KUKA KRL program: EPS_2_25694_HR03_A_20260120031654.src

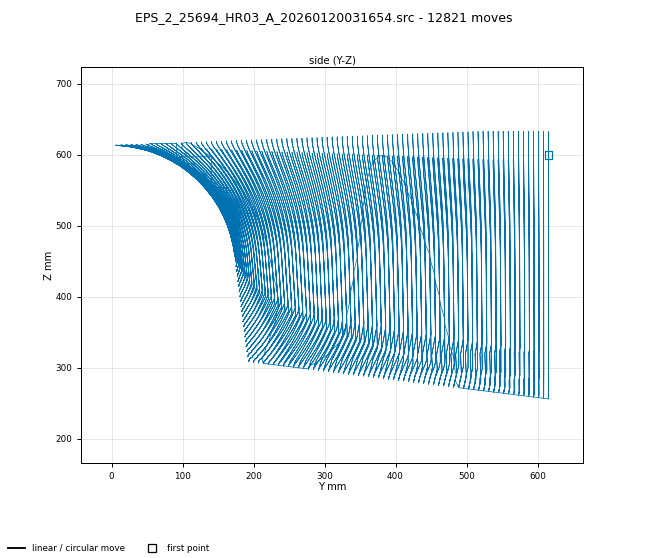
[picture p0: tool path of EPS_2_25694_HR03_A_20260120031654.src, 12821 of 12823 moves have a stored position in this frame; points joined in program order, loops and branches not executed]
&ACCESS RVP
&REL 4
&COMMENT QRS 19112012
&PARAM EDITMASK = *
DEF PART()
EXT BAS (BAS_COMMAND :IN,REAL :IN )
INT I
BAS (#INITMOV,0 )

;KUKA QRS Post kuka4.cps  Date:22-06-2017 !

File_ID=2992

QRS_PRE_INIT()

;Init var - Until changes are made in qrs_pre_init
Outlet_Square_prg=0
Inlet_1_Square_prg=0
Inlet_2_Square_prg=0
Inlet_3_Square_prg=0
Inlet_4_Square_prg=0
Inlet_5_Square_prg=0

Outlet_1={X 0.000, Y 523.550, Z 484.000, B 0.000, E1 0.000 }
Inlet_1={X 0.000, Y 526.470, Z 444.000, B 0.000, E1 180.000 }
Outlet_1_type=299
Inlet_1_type=299
;QRS#1=Sidecore dimensions
;QRS#2=300-12" PVC SDR 35
;QRS#3=300-12" PVC SDR 35
;QRS#4=
;QRS#5=
;QRS#6=
;QRS#7=
;QRS#8=
;QRS#9=16M PSX
;QRS#10=16M PSX
;QRS#11=
;QRS#12=
;QRS#13=
;QRS#14=
;QRS#15=
;QRS#16=1220x127x914 3'
;QRS#17=EPS Height
;QRS#18=633,5
;QRS#19=*
;QRS#20= UPDATED VERSION 22-06-2017
;QRS#21=*
Outlet_Square=0150
Inlet_1_Square=0150
Inlet_2_Square=0
Inlet_3_Square=0
Inlet_4_Square=0
Inlet_5_Square=0
Mill_Square=1
Outlet_Square_Prg=206
Inlet_1_Square_prg=206

QRS_INIT()

$ADVANCE=5

; T1
PTP {E1 173.656,E2 173.656}
PTP {X 0,Y 615.44,A -85,B 0,C 180,E1 173.656,E2 173.656,E3 0,E4 0,E5 0,E6 0}
QRS_SPEED_INIT()
LIN {X 0,Y 615.44,Z 600,A -85,B 0,C 180,E1 173.656,E2 173.656,E3 0,E4 0,E5 0,E6 0} C_VEL
LIN {X 0,Y 615.44,Z 266.5,A -85,B 0,C 180,E1 173.656,E2 173.656} C_VEL
LIN {X 0,Y 615.44,Z 258.32,A -85,B 0,C 180,E1 173.656,E2 173.656} C_VEL
LIN {X 0,Y 615.434,Z 256.32,A -85,B 0,C 180,E1 173.47,E2 173.47} C_VEL
LIN {X 0,Y 615.463,Z 256.318,A -85,B 0,C 180,E1 170.801,E2 170.801} C_VEL
LIN {X 0,Y 615.474,Z 256.325,A -85,B 0,C 180,E1 168.139,E2 168.139} C_VEL
LIN {X 0,Y 615.429,Z 256.321,A -85,B 0,C 180,E1 165.449,E2 165.449} C_VEL
LIN {X 0,Y 615.48,Z 256.318,A -85,B 0,C 180,E1 162.729,E2 162.729} C_VEL
LIN {X 0,Y 615.445,Z 256.323,A -85,B 0,C 180,E1 159.966,E2 159.966} C_VEL
LIN {X 0,Y 615.426,Z 256.322,A -85,B 0,C 180,E1 157.669,E2 157.669} C_VEL
LIN {X 0,Y 615.425,Z 256.323,A -85,B 0,C 180,E1 155.725,E2 155.725} C_VEL
LIN {X 0,Y 615.423,Z 256.322,A -85,B 0,C 180,E1 153.553,E2 153.553} C_VEL
LIN {X 0,Y 615.493,Z 256.324,A -85,B 0,C 180,E1 150.594,E2 150.594} C_VEL
LIN {X 0,Y 615.465,Z 256.324,A -85,B 0,C 180,E1 148.313,E2 148.313} C_VEL
LIN {X 0,Y 615.429,Z 256.324,A -85,B 0,C 180,E1 145.974,E2 145.974} C_VEL
LIN {X 0,Y 615.418,Z 256.323,A -85,B 0,C 180,E1 143.57,E2 143.57} C_VEL
LIN {X 0,Y 615.463,Z 256.323,A -85,B 0,C 180,E1 140.942,E2 140.942} C_VEL
LIN {X 0,Y 615.473,Z 256.326,A -85,B 0,C 180,E1 138.525,E2 138.525} C_VEL
LIN {X 0,Y 615.42,Z 256.325,A -85,B 0,C 180,E1 136.01,E2 136.01} C_VEL
LIN {X 0,Y 615.417,Z 256.325,A -85,B 0,C 180,E1 133.99,E2 133.99} C_VEL
LIN {X 0,Y 615.417,Z 256.325,A -85,B 0,C 180,E1 131.48,E2 131.48} C_VEL
LIN {X 0,Y 615.473,Z 256.327,A -85,B 0,C 180,E1 128.906,E2 128.906} C_VEL
LIN {X 0,Y 615.446,Z 256.324,A -85,B 0,C 180,E1 126.428,E2 126.428} C_VEL
LIN {X 0,Y 615.416,Z 256.324,A -85,B 0,C 180,E1 124.027,E2 124.027} C_VEL
LIN {X 0,Y 615.415,Z 256.325,A -85,B 0,C 180,E1 121.69,E2 121.69} C_VEL
LIN {X 0,Y 615.435,Z 256.324,A -85,B 0,C 180,E1 119.41,E2 119.41} C_VEL
LIN {X 0,Y 615.445,Z 256.322,A -85,B 0,C 180,E1 116.447,E2 116.447} C_VEL
LIN {X 0,Y 615.419,Z 256.323,A -85,B 0,C 180,E1 113.994,E2 113.994} C_VEL
LIN {X 0,Y 615.424,Z 256.408,A -85,B 0,C 180,E1 111.72,E2 111.72} C_VEL
LIN {X 0,Y 615.484,Z 275.615,A -85,B 0,C 180,E1 109.165,E2 109.165} C_VEL
LIN {X 0,Y 615.468,Z 283.1,A -85,B 0,C 180,E1 108.181,E2 108.181} C_VEL
LIN {X 0,Y 615.489,Z 447.324,A -85,B 0,C 180,E1 106.2,E2 106.2} C_VEL
LIN {X 0,Y 615.489,Z 461.801,A -85,B 0,C 180,E1 105.906,E2 105.906} C_VEL
LIN {X 0,Y 615.477,Z 476.406,A -85,B 0,C 180,E1 105.481,E2 105.481} C_VEL
LIN {X 0,Y 615.491,Z 489.73,A -85,B 0,C 180,E1 104.972,E2 104.972} C_VEL
LIN {X 0,Y 615.483,Z 503.376,A -85,B 0,C 180,E1 104.32,E2 104.32} C_VEL
LIN {X 0,Y 615.5,Z 516.661,A -85,B 0,C 180,E1 103.538,E2 103.538} C_VEL
LIN {X 0,Y 615.497,Z 528.512,A -85,B 0,C 180,E1 102.698,E2 102.698} C_VEL
LIN {X 0,Y 615.497,Z 540.356,A -85,B 0,C 180,E1 101.694,E2 101.694} C_VEL
LIN {X 0,Y 615.495,Z 550.165,A -85,B 0,C 180,E1 100.709,E2 100.709} C_VEL
LIN {X 0,Y 615.495,Z 560.01,A -85,B 0,C 180,E1 99.531,E2 99.531} C_VEL
LIN {X 0,Y 615.497,Z 568.101,A -85,B 0,C 180,E1 98.371,E2 98.371} C_VEL
LIN {X 0,Y 615.491,Z 574.781,A -85,B 0,C 180,E1 97.216,E2 97.216} C_VEL
LIN {X 0,Y 615.497,Z 580.947,A -85,B 0,C 180,E1 95.899,E2 95.899} C_VEL
LIN {X 0,Y 615.49,Z 585.715,A -85,B 0,C 180,E1 94.585,E2 94.585} C_VEL
LIN {X 0,Y 615.491,Z 589.22,A -85,B 0,C 180,E1 93.273,E2 93.273} C_VEL
LIN {X 0,Y 615.499,Z 591.539,A -85,B 0,C 180,E1 91.963,E2 91.963} C_VEL
LIN {X 0,Y 615.491,Z 592.728,A -85,B 0,C 180,E1 90.655,E2 90.655} C_VEL
LIN {X 0,Y 615.492,Z 592.751,A -85,B 0,C 180,E1 89.346,E2 89.346} C_VEL
LIN {X 0,Y 615.499,Z 591.646,A -85,B 0,C 180,E1 88.037,E2 88.037} C_VEL
LIN {X 0,Y 615.494,Z 589.416,A -85,B 0,C 180,E1 86.727,E2 86.727} C_VEL
LIN {X 0,Y 615.491,Z 586.006,A -85,B 0,C 180,E1 85.416,E2 85.416} C_VEL
LIN {X 0,Y 615.498,Z 581.337,A -85,B 0,C 180,E1 84.102,E2 84.102} C_VEL
LIN {X 0,Y 615.49,Z 575.273,A -85,B 0,C 180,E1 82.785,E2 82.785} C_VEL
LIN {X 0,Y 615.49,Z 567.635,A -85,B 0,C 180,E1 81.464,E2 81.464} C_VEL
LIN {X 0,Y 615.495,Z 559.452,A -85,B 0,C 180,E1 80.304,E2 80.304} C_VEL
LIN {X 0,Y 615.496,Z 549.333,A -85,B 0,C 180,E1 79.109,E2 79.109} C_VEL
LIN {X 0,Y 615.498,Z 537.685,A -85,B 0,C 180,E1 77.973,E2 77.973} C_VEL
LIN {X 0,Y 615.498,Z 526.415,A -85,B 0,C 180,E1 77.051,E2 77.051} C_VEL
LIN {X 0,Y 615.498,Z 514.177,A -85,B 0,C 180,E1 76.211,E2 76.211} C_VEL
LIN {X 0,Y 615.48,Z 500.78,A -85,B 0,C 180,E1 75.451,E2 75.451} C_VEL
LIN {X 0,Y 615.488,Z 485.866,A -85,B 0,C 180,E1 74.774,E2 74.774} C_VEL
LIN {X 0,Y 615.477,Z 471.391,A -85,B 0,C 180,E1 74.265,E2 74.265} C_VEL
LIN {X 0,Y 615.491,Z 455.809,A -85,B 0,C 180,E1 73.866,E2 73.866} C_VEL
LIN {X 0,Y 615.486,Z 439.601,A -85,B 0,C 180,E1 73.603,E2 73.603} C_VEL
LIN {X 0,Y 615.472,Z 283.019,A -85,B 0,C 180,E1 71.718,E2 71.718} C_VEL
LIN {X 0,Y 615.498,Z 261.851,A -85,B 0,C 180,E1 68.92,E2 68.92} C_VEL
LIN {X 0,Y 615.43,Z 256.322,A -85,B 0,C 180,E1 68.17,E2 68.17} C_VEL
LIN {X 0,Y 615.434,Z 256.32,A -85,B 0,C 180,E1 65.726,E2 65.726} C_VEL
LIN {X 0,Y 615.494,Z 256.326,A -85,B 0,C 180,E1 62.954,E2 62.954} C_VEL
LIN {X 0,Y 615.423,Z 256.323,A -85,B 0,C 180,E1 60.216,E2 60.216} C_VEL
LIN {X 0,Y 615.425,Z 256.323,A -85,B 0,C 180,E1 58.311,E2 58.311} C_VEL
LIN {X 0,Y 615.422,Z 256.322,A -85,B 0,C 180,E1 55.974,E2 55.974} C_VEL
LIN {X 0,Y 615.449,Z 256.322,A -85,B 0,C 180,E1 53.573,E2 53.573} C_VEL
LIN {X 0,Y 615.47,Z 256.325,A -85,B 0,C 180,E1 50.94,E2 50.94} C_VEL
LIN {X 0,Y 615.425,Z 256.324,A -85,B 0,C 180,E1 48.521,E2 48.521} C_VEL
LIN {X 0,Y 615.417,Z 256.324,A -85,B 0,C 180,E1 46.009,E2 46.009} C_VEL
LIN {X 0,Y 615.498,Z 256.325,A -85,B 0,C 180,E1 43.244,E2 43.244} C_VEL
LIN {X 0,Y 615.42,Z 256.325,A -85,B 0,C 180,E1 40.612,E2 40.612} C_VEL
LIN {X 0,Y 615.418,Z 256.325,A -85,B 0,C 180,E1 38.004,E2 38.004} C_VEL
LIN {X 0,Y 615.456,Z 256.325,A -85,B 0,C 180,E1 35.618,E2 35.618} C_VEL
LIN {X 0,Y 615.483,Z 256.324,A -85,B 0,C 180,E1 33.237,E2 33.237} C_VEL
LIN {X 0,Y 615.444,Z 256.323,A -85,B 0,C 180,E1 30.922,E2 30.922} C_VEL
LIN {X 0,Y 615.416,Z 256.323,A -85,B 0,C 180,E1 28.438,E2 28.438} C_VEL
LIN {X 0,Y 615.418,Z 256.323,A -85,B 0,C 180,E1 26.447,E2 26.447} C_VEL
LIN {X 0,Y 615.435,Z 256.324,A -85,B 0,C 180,E1 23.998,E2 23.998} C_VEL
LIN {X 0,Y 615.498,Z 256.322,A -85,B 0,C 180,E1 21.432,E2 21.432} C_VEL
LIN {X 0,Y 615.424,Z 256.322,A -85,B 0,C 180,E1 18.587,E2 18.587} C_VEL
LIN {X 0,Y 615.424,Z 256.322,A -85,B 0,C 180,E1 16.412,E2 16.412} C_VEL
LIN {X 0,Y 615.461,Z 256.325,A -85,B 0,C 180,E1 13.875,E2 13.875} C_VEL
LIN {X 0,Y 615.466,Z 256.318,A -85,B 0,C 180,E1 11.194,E2 11.194} C_VEL
LIN {X 0,Y 615.429,Z 256.321,A -85,B 0,C 180,E1 8.538,E2 8.538} C_VEL
LIN {X 0,Y 615.475,Z 256.324,A -85,B 0,C 180,E1 5.899,E2 5.899} C_VEL
LIN {X 0,Y 615.471,Z 256.317,A -85,B 0,C 180,E1 3.273,E2 3.273} C_VEL
LIN {X 0,Y 615.433,Z 256.32,A -85,B 0,C 180,E1 0.654,E2 0.654} C_VEL
LIN {X 0,Y 615.471,Z 256.324,A -85,B 0,C 180,E1 -1.963,E2 -1.963} C_VEL
LIN {X 0,Y 615.485,Z 256.314,A -85,B 0,C 180,E1 -4.584,E2 -4.584} C_VEL
LIN {X 0,Y 615.438,Z 256.319,A -85,B 0,C 180,E1 -7.216,E2 -7.216} C_VEL
LIN {X 0,Y 615.472,Z 256.324,A -85,B 0,C 180,E1 -9.862,E2 -9.862} C_VEL
LIN {X 0,Y 615.48,Z 256.314,A -85,B 0,C 180,E1 -12.53,E2 -12.53} C_VEL
LIN {X 0,Y 615.441,Z 256.319,A -85,B 0,C 180,E1 -15.227,E2 -15.227} C_VEL
LIN {X 0,Y 615.493,Z 256.326,A -85,B 0,C 180,E1 -17.957,E2 -17.957} C_VEL
LIN {X 0,Y 615.462,Z 256.314,A -85,B 0,C 180,E1 -20.732,E2 -20.732} C_VEL
LIN {X 0,Y 615.454,Z 256.315,A -85,B 0,C 180,E1 -22.846,E2 -22.846} C_VEL
LIN {X 0,Y 615.449,Z 256.316,A -85,B 0,C 180,E1 -24.993,E2 -24.993} C_VEL
LIN {X 0,Y 615.449,Z 256.318,A -85,B 0,C 180,E1 -27.179,E2 -27.179} C_VEL
LIN {X 0,Y 615.498,Z 256.325,A -85,B 0,C 180,E1 -29.797,E2 -29.797} C_VEL
LIN {X 0,Y 615.484,Z 256.31,A -85,B 0,C 180,E1 -32.458,E2 -32.458} C_VEL
LIN {X 0,Y 615.457,Z 256.314,A -85,B 0,C 180,E1 -34.817,E2 -34.817} C_VEL
LIN {X 0,Y 615.458,Z 256.32,A -85,B 0,C 180,E1 -37.244,E2 -37.244} C_VEL
LIN {X 0,Y 615.493,Z 256.313,A -85,B 0,C 180,E1 -40.09,E2 -40.09} C_VEL
LIN {X 0,Y 615.49,Z 256.309,A -85,B 0,C 180,E1 -42.353,E2 -42.353} C_VEL
LIN {X 0,Y 615.459,Z 256.318,A -85,B 0,C 180,E1 -45.071,E2 -45.071} C_VEL
LIN {X 0,Y 615.49,Z 256.316,A -85,B 0,C 180,E1 -47.919,E2 -47.919} C_VEL
LIN {X 0,Y 615.493,Z 256.308,A -85,B 0,C 180,E1 -50.251,E2 -50.251} C_VEL
LIN {X 0,Y 615.465,Z 256.319,A -85,B 0,C 180,E1 -53.066,E2 -53.066} C_VEL
LIN {X 0,Y 615.482,Z 256.322,A -85,B 0,C 180,E1 -55.3,E2 -55.3} C_VEL
LIN {X 0,Y 615.483,Z 256.309,A -85,B 0,C 180,E1 -58.315,E2 -58.315} C_VEL
LIN {X 0,Y 615.468,Z 256.312,A -85,B 0,C 180,E1 -60.593,E2 -60.593} C_VEL
LIN {X 0,Y 615.469,Z 256.318,A -85,B 0,C 180,E1 -62.958,E2 -62.958} C_VEL
LIN {X 0,Y 615.47,Z 256.455,A -85,B 0,C 180,E1 -64.541,E2 -64.541} C_VEL
LIN {X 0,Y 615.483,Z 280.841,A -85,B 0,C 180,E1 -67.28,E2 -67.28} C_VEL
LIN {X 0,Y 615.494,Z 305.255,A -85,B 0,C 180,E1 -69.968,E2 -69.968} C_VEL
LIN {X 0,Y 615.499,Z 322.022,A -85,B 0,C 180,E1 -71.762,E2 -71.762} C_VEL
LIN {X 0,Y 615.487,Z 488.125,A -85,B 0,C 180,E1 -73.767,E2 -73.767} C_VEL
LIN {X 0,Y 615.49,Z 503.724,A -85,B 0,C 180,E1 -74.095,E2 -74.095} C_VEL
LIN {X 0,Y 615.48,Z 519.059,A -85,B 0,C 180,E1 -74.562,E2 -74.562} C_VEL
LIN {X 0,Y 615.492,Z 532.76,A -85,B 0,C 180,E1 -75.113,E2 -75.113} C_VEL
LIN {X 0,Y 615.494,Z 547.048,A -85,B 0,C 180,E1 -75.834,E2 -75.834} C_VEL
LIN {X 0,Y 615.497,Z 559.903,A -85,B 0,C 180,E1 -76.631,E2 -76.631} C_VEL
LIN {X 0,Y 615.495,Z 572.259,A -85,B 0,C 180,E1 -77.554,E2 -77.554} C_VEL
LIN {X 0,Y 615.495,Z 582.61,A -85,B 0,C 180,E1 -78.474,E2 -78.474} C_VEL
LIN {X 0,Y 615.495,Z 592.187,A -85,B 0,C 180,E1 -79.473,E2 -79.473} C_VEL
LIN {X 0,Y 615.494,Z 601.579,A -85,B 0,C 180,E1 -80.636,E2 -80.636} C_VEL
LIN {X 0,Y 615.495,Z 609.383,A -85,B 0,C 180,E1 -81.794,E2 -81.794} C_VEL
LIN {X 0,Y 615.496,Z 616.607,A -85,B 0,C 180,E1 -83.102,E2 -83.102} C_VEL
LIN {X 0,Y 615.499,Z 622.438,A -85,B 0,C 180,E1 -84.431,E2 -84.431} C_VEL
LIN {X 0,Y 615.491,Z 625.861,A -85,B 0,C 180,E1 -85.416,E2 -85.416} C_VEL
LIN {X 0,Y 615.492,Z 629.319,A -85,B 0,C 180,E1 -86.727,E2 -86.727} C_VEL
LIN {X 0,Y 615.497,Z 631.594,A -85,B 0,C 180,E1 -88.037,E2 -88.037} C_VEL
LIN {X 0,Y 615.493,Z 632.741,A -85,B 0,C 180,E1 -89.346,E2 -89.346} C_VEL
LIN {X 0,Y 615.493,Z 632.74,A -85,B 0,C 180,E1 -90.655,E2 -90.655} C_VEL
LIN {X 0,Y 615.497,Z 631.593,A -85,B 0,C 180,E1 -91.963,E2 -91.963} C_VEL
LIN {X 0,Y 615.492,Z 629.317,A -85,B 0,C 180,E1 -93.273,E2 -93.273} C_VEL
LIN {X 0,Y 615.491,Z 625.859,A -85,B 0,C 180,E1 -94.585,E2 -94.585} C_VEL
LIN {X 0,Y 615.49,Z 621.142,A -85,B 0,C 180,E1 -95.899,E2 -95.899} C_VEL
LIN {X 0,Y 615.495,Z 615.027,A -85,B 0,C 180,E1 -97.216,E2 -97.216} C_VEL
LIN {X 0,Y 615.49,Z 607.331,A -85,B 0,C 180,E1 -98.537,E2 -98.537} C_VEL
LIN {X 0,Y 615.495,Z 599.111,A -85,B 0,C 180,E1 -99.696,E2 -99.696} C_VEL
LIN {X 0,Y 615.497,Z 588.895,A -85,B 0,C 180,E1 -100.893,E2 -100.893} C_VEL
LIN {X 0,Y 615.495,Z 579.063,A -85,B 0,C 180,E1 -101.861,E2 -101.861} C_VEL
LIN {X 0,Y 615.498,Z 566.942,A -85,B 0,C 180,E1 -102.866,E2 -102.866} C_VEL
LIN {X 0,Y 615.498,Z 554.792,A -85,B 0,C 180,E1 -103.706,E2 -103.706} C_VEL
LIN {X 0,Y 615.484,Z 541.372,A -85,B 0,C 180,E1 -104.473,E2 -104.473} C_VEL
LIN {X 0,Y 615.495,Z 526.839,A -85,B 0,C 180,E1 -105.141,E2 -105.141} C_VEL
LIN {X 0,Y 615.484,Z 512.604,A -85,B 0,C 180,E1 -105.651,E2 -105.651} C_VEL
LIN {X 0,Y 615.499,Z 498.113,A -85,B 0,C 180,E1 -106.036,E2 -106.036} C_VEL
LIN {X 0,Y 615.487,Z 483.525,A -85,B 0,C 180,E1 -106.298,E2 -106.298} C_VEL
LIN {X 0,Y 615.497,Z 321.596,A -85,B 0,C 180,E1 -108.259,E2 -108.259} C_VEL
LIN {X 0,Y 615.476,Z 295.674,A -85,B 0,C 180,E1 -111.082,E2 -111.082} C_VEL
LIN {X 0,Y 615.495,Z 271.314,A -85,B 0,C 180,E1 -113.782,E2 -113.782} C_VEL
LIN {X 0,Y 615.472,Z 256.311,A -85,B 0,C 180,E1 -115.495,E2 -115.495} C_VEL
LIN {X 0,Y 615.49,Z 256.322,A -85,B 0,C 180,E1 -118.451,E2 -118.451} C_VEL
LIN {X 0,Y 615.464,Z 256.318,A -85,B 0,C 180,E1 -121.082,E2 -121.082} C_VEL
LIN {X 0,Y 615.475,Z 256.31,A -85,B 0,C 180,E1 -123.532,E2 -123.532} C_VEL
LIN {X 0,Y 615.485,Z 256.326,A -85,B 0,C 180,E1 -126.425,E2 -126.425} C_VEL
LIN {X 0,Y 615.461,Z 256.317,A -85,B 0,C 180,E1 -129.059,E2 -129.059} C_VEL
LIN {X 0,Y 615.472,Z 256.311,A -85,B 0,C 180,E1 -131.476,E2 -131.476} C_VEL
LIN {X 0,Y 615.488,Z 256.319,A -85,B 0,C 180,E1 -134.15,E2 -134.15} C_VEL
LIN {X 0,Y 615.466,Z 256.32,A -85,B 0,C 180,E1 -136.754,E2 -136.754} C_VEL
LIN {X 0,Y 615.468,Z 256.312,A -85,B 0,C 180,E1 -139.392,E2 -139.392} C_VEL
LIN {X 0,Y 615.49,Z 256.316,A -85,B 0,C 180,E1 -141.989,E2 -141.989} C_VEL
LIN {X 0,Y 615.488,Z 256.324,A -85,B 0,C 180,E1 -144.384,E2 -144.384} C_VEL
LIN {X 0,Y 615.457,Z 256.319,A -85,B 0,C 180,E1 -146.762,E2 -146.762} C_VEL
LIN {X 0,Y 615.454,Z 256.315,A -85,B 0,C 180,E1 -149.078,E2 -149.078} C_VEL
LIN {X 0,Y 615.487,Z 256.31,A -85,B 0,C 180,E1 -151.551,E2 -151.551} C_VEL
LIN {X 0,Y 615.469,Z 256.322,A -85,B 0,C 180,E1 -154.436,E2 -154.436} C_VEL
LIN {X 0,Y 615.466,Z 256.322,A -85,B 0,C 180,E1 -156.443,E2 -156.443} C_VEL
LIN {X 0,Y 615.456,Z 256.32,A -85,B 0,C 180,E1 -158.567,E2 -158.567} C_VEL
LIN {X 0,Y 615.45,Z 256.319,A -85,B 0,C 180,E1 -160.661,E2 -160.661} C_VEL
LIN {X 0,Y 615.446,Z 256.319,A -85,B 0,C 180,E1 -162.728,E2 -162.728} C_VEL
LIN {X 0,Y 615.483,Z 256.312,A -85,B 0,C 180,E1 -165.451,E2 -165.451} C_VEL
LIN {X 0,Y 615.48,Z 256.324,A -85,B 0,C 180,E1 -168.139,E2 -168.139} C_VEL
LIN {X 0,Y 615.442,Z 256.318,A -85,B 0,C 180,E1 -170.801,E2 -170.801} C_VEL
LIN {X 0,Y 615.487,Z 256.313,A -85,B 0,C 180,E1 -173.443,E2 -173.443} C_VEL
LIN {X 0,Y 615.476,Z 256.324,A -85,B 0,C 180,E1 -176.071,E2 -176.071} C_VEL
LIN {X 0,Y 615.438,Z 256.319,A -85,B 0,C 180,E1 -178.691,E2 -178.691} C_VEL
LIN {X 0,Y 615.475,Z 256.315,A -85,B 0,C 180,E1 -181.309,E2 -181.309} C_VEL
LIN {X 0,Y 615.477,Z 256.325,A -85,B 0,C 180,E1 -183.929,E2 -183.929} C_VEL
LIN {X 0,Y 615.434,Z 256.32,A -85,B 0,C 180,E1 -186.53,E2 -186.53} C_VEL
LIN {X 0,Y 614.778,Z 256.465,A -85,B 0,C 180,E1 -187.076,E2 -187.076} C_VEL
LIN {X 0,Y 611.96,Z 256.882,A -85,B 0,C 180,E1 -187.962,E2 -187.962} C_VEL
LIN {X 0,Y 609.571,Z 257.191,A -85,B 0,C 180,E1 -188.675,E2 -188.675} C_VEL
LIN {X 0,Y 608.534,Z 257.307,A -85,B 0,C 180,E1 -189.225,E2 -189.225} C_VEL
LIN {X 0,Y 608.444,Z 257.317,A -85,B 0,C 180,E1 -189.411,E2 -189.411} C_VEL
LIN {X 0,Y 608.443,Z 257.319,A -85,B 0,C 180,E1 -192,E2 -192} C_VEL
LIN {X 0,Y 608.405,Z 257.318,A -85,B 0,C 180,E1 -194.722,E2 -194.722} C_VEL
LIN {X 0,Y 608.44,Z 257.322,A -85,B 0,C 180,E1 -197.477,E2 -197.477} C_VEL
LIN {X 0,Y 608.416,Z 257.318,A -85,B 0,C 180,E1 -200.276,E2 -200.276} C_VEL
LIN {X 0,Y 608.397,Z 257.319,A -85,B 0,C 180,E1 -202.461,E2 -202.461} C_VEL
LIN {X 0,Y 608.411,Z 257.318,A -85,B 0,C 180,E1 -204.573,E2 -204.573} C_VEL
LIN {X 0,Y 608.463,Z 257.316,A -85,B 0,C 180,E1 -207.203,E2 -207.203} C_VEL
LIN {X 0,Y 608.412,Z 257.32,A -85,B 0,C 180,E1 -209.961,E2 -209.961} C_VEL
LIN {X 0,Y 608.405,Z 257.318,A -85,B 0,C 180,E1 -212.513,E2 -212.513} C_VEL
LIN {X 0,Y 608.406,Z 257.321,A -85,B 0,C 180,E1 -214.899,E2 -214.899} C_VEL
LIN {X 0,Y 608.432,Z 257.319,A -85,B 0,C 180,E1 -217.749,E2 -217.749} C_VEL
LIN {X 0,Y 608.405,Z 257.318,A -85,B 0,C 180,E1 -220.323,E2 -220.323} C_VEL
LIN {X 0,Y 608.426,Z 257.32,A -85,B 0,C 180,E1 -222.962,E2 -222.962} C_VEL
LIN {X 0,Y 608.407,Z 257.321,A -85,B 0,C 180,E1 -225.741,E2 -225.741} C_VEL
LIN {X 0,Y 608.405,Z 257.319,A -85,B 0,C 180,E1 -227.933,E2 -227.933} C_VEL
LIN {X 0,Y 608.413,Z 257.32,A -85,B 0,C 180,E1 -230.709,E2 -230.709} C_VEL
LIN {X 0,Y 608.435,Z 257.324,A -85,B 0,C 180,E1 -233.083,E2 -233.083} C_VEL
LIN {X 0,Y 608.448,Z 257.317,A -85,B 0,C 180,E1 -235.529,E2 -235.529} C_VEL
LIN {X 0,Y 608.414,Z 257.318,A -85,B 0,C 180,E1 -237.902,E2 -237.902} C_VEL
LIN {X 0,Y 608.404,Z 257.319,A -85,B 0,C 180,E1 -240.217,E2 -240.217} C_VEL
LIN {X 0,Y 608.441,Z 257.32,A -85,B 0,C 180,E1 -242.8,E2 -242.8} C_VEL
LIN {X 0,Y 608.428,Z 257.32,A -85,B 0,C 180,E1 -245.427,E2 -245.427} C_VEL
LIN {X 0,Y 608.428,Z 257.399,A -85,B 0,C 180,E1 -248.151,E2 -248.151} C_VEL
LIN {X 0,Y 608.549,Z 271.691,A -85,B 0,C 180,E1 -250.081,E2 -250.081} C_VEL
LIN {X 0,Y 608.517,Z 283.131,A -85,B 0,C 180,E1 -251.604,E2 -251.604} C_VEL
LIN {X 0,Y 608.727,Z 300.004,A -85,B 0,C 180,E1 -251.816,E2 -251.816} C_VEL
LIN {X 0,Y 608.684,Z 448.405,A -85,B 0,C 180,E1 -253.631,E2 -253.631} C_VEL
LIN {X 0,Y 608.648,Z 463.624,A -85,B 0,C 180,E1 -253.954,E2 -253.954} C_VEL
LIN {X 0,Y 608.61,Z 478.983,A -85,B 0,C 180,E1 -254.426,E2 -254.426} C_VEL
LIN {X 0,Y 608.59,Z 493.666,A -85,B 0,C 180,E1 -255.025,E2 -255.025} C_VEL
LIN {X 0,Y 608.571,Z 507.434,A -85,B 0,C 180,E1 -255.734,E2 -255.734} C_VEL
LIN {X 0,Y 608.548,Z 520.538,A -85,B 0,C 180,E1 -256.56,E2 -256.56} C_VEL
LIN {X 0,Y 608.505,Z 532.836,A -85,B 0,C 180,E1 -257.493,E2 -257.493} C_VEL
LIN {X 0,Y 608.498,Z 544.047,A -85,B 0,C 180,E1 -258.508,E2 -258.508} C_VEL
LIN {X 0,Y 608.477,Z 554.932,A -85,B 0,C 180,E1 -259.687,E2 -259.687} C_VEL
LIN {X 0,Y 608.469,Z 563.982,A -85,B 0,C 180,E1 -260.861,E2 -260.861} C_VEL
LIN {X 0,Y 608.459,Z 571.478,A -85,B 0,C 180,E1 -262.032,E2 -262.032} C_VEL
LIN {X 0,Y 608.445,Z 578.628,A -85,B 0,C 180,E1 -263.396,E2 -263.396} C_VEL
LIN {X 0,Y 608.436,Z 583.992,A -85,B 0,C 180,E1 -264.698,E2 -264.698} C_VEL
LIN {X 0,Y 608.432,Z 588.166,A -85,B 0,C 180,E1 -266.026,E2 -266.026} C_VEL
LIN {X 0,Y 608.421,Z 591.109,A -85,B 0,C 180,E1 -267.351,E2 -267.351} C_VEL
LIN {X 0,Y 608.444,Z 592.88,A -85,B 0,C 180,E1 -268.676,E2 -268.676} C_VEL
LIN {X 0,Y 608.432,Z 593.495,A -85,B 0,C 180,E1 -270,E2 -270} C_VEL
LIN {X 0,Y 608.446,Z 592.944,A -85,B 0,C 180,E1 -271.323,E2 -271.323} C_VEL
LIN {X 0,Y 608.424,Z 591.26,A -85,B 0,C 180,E1 -272.648,E2 -272.648} C_VEL
LIN {X 0,Y 608.432,Z 588.409,A -85,B 0,C 180,E1 -273.974,E2 -273.974} C_VEL
LIN {X 0,Y 608.436,Z 584.33,A -85,B 0,C 180,E1 -275.302,E2 -275.302} C_VEL
LIN {X 0,Y 608.445,Z 578.923,A -85,B 0,C 180,E1 -276.633,E2 -276.633} C_VEL
LIN {X 0,Y 608.457,Z 572.025,A -85,B 0,C 180,E1 -277.967,E2 -277.967} C_VEL
LIN {X 0,Y 608.466,Z 564.593,A -85,B 0,C 180,E1 -279.138,E2 -279.138} C_VEL
LIN {X 0,Y 608.476,Z 555.665,A -85,B 0,C 180,E1 -280.313,E2 -280.313} C_VEL
LIN {X 0,Y 608.496,Z 544.949,A -85,B 0,C 180,E1 -281.492,E2 -281.492} C_VEL
LIN {X 0,Y 608.513,Z 532.909,A -85,B 0,C 180,E1 -282.591,E2 -282.591} C_VEL
LIN {X 0,Y 608.543,Z 520.621,A -85,B 0,C 180,E1 -283.524,E2 -283.524} C_VEL
LIN {X 0,Y 608.584,Z 507.68,A -85,B 0,C 180,E1 -284.342,E2 -284.342} C_VEL
LIN {X 0,Y 608.606,Z 493.775,A -85,B 0,C 180,E1 -285.059,E2 -285.059} C_VEL
LIN {X 0,Y 608.627,Z 479.113,A -85,B 0,C 180,E1 -285.659,E2 -285.659} C_VEL
LIN {X 0,Y 608.662,Z 463.541,A -85,B 0,C 180,E1 -286.138,E2 -286.138} C_VEL
LIN {X 0,Y 608.687,Z 447.541,A -85,B 0,C 180,E1 -286.473,E2 -286.473} C_VEL
LIN {X 0,Y 608.637,Z 283.846,A -85,B 0,C 180,E1 -288.474,E2 -288.474} C_VEL
LIN {X 0,Y 608.533,Z 283.04,A -85,B 0,C 180,E1 -288.498,E2 -288.498} C_VEL
LIN {X 0,Y 608.592,Z 263.164,A -85,B 0,C 180,E1 -291.154,E2 -291.154} C_VEL
LIN {X 0,Y 608.41,Z 257.32,A -85,B 0,C 180,E1 -291.961,E2 -291.961} C_VEL
LIN {X 0,Y 608.433,Z 257.318,A -85,B 0,C 180,E1 -294.572,E2 -294.572} C_VEL
LIN {X 0,Y 608.421,Z 257.319,A -85,B 0,C 180,E1 -297.519,E2 -297.519} C_VEL
LIN {X 0,Y 608.394,Z 257.32,A -85,B 0,C 180,E1 -299.959,E2 -299.959} C_VEL
LIN {X 0,Y 608.432,Z 257.319,A -85,B 0,C 180,E1 -302.518,E2 -302.518} C_VEL
LIN {X 0,Y 608.414,Z 257.322,A -85,B 0,C 180,E1 -305.279,E2 -305.279} C_VEL
LIN {X 0,Y 608.397,Z 257.319,A -85,B 0,C 180,E1 -307.751,E2 -307.751} C_VEL
LIN {X 0,Y 608.432,Z 257.317,A -85,B 0,C 180,E1 -310.327,E2 -310.327} C_VEL
LIN {X 0,Y 608.433,Z 257.318,A -85,B 0,C 180,E1 -313.305,E2 -313.305} C_VEL
LIN {X 0,Y 608.416,Z 257.318,A -85,B 0,C 180,E1 -316.126,E2 -316.126} C_VEL
LIN {X 0,Y 608.436,Z 257.324,A -85,B 0,C 180,E1 -318.822,E2 -318.822} C_VEL
LIN {X 0,Y 608.392,Z 257.321,A -85,B 0,C 180,E1 -321.406,E2 -321.406} C_VEL
LIN {X 0,Y 608.416,Z 257.32,A -85,B 0,C 180,E1 -323.082,E2 -323.082} C_VEL
LIN {X 0,Y 608.412,Z 257.317,A -85,B 0,C 180,E1 -325.527,E2 -325.527} C_VEL
LIN {X 0,Y 608.413,Z 257.318,A -85,B 0,C 180,E1 -327.902,E2 -327.902} C_VEL
LIN {X 0,Y 608.432,Z 257.319,A -85,B 0,C 180,E1 -330.218,E2 -330.218} C_VEL
LIN {X 0,Y 608.401,Z 257.32,A -85,B 0,C 180,E1 -333.223,E2 -333.223} C_VEL
LIN {X 0,Y 608.406,Z 257.318,A -85,B 0,C 180,E1 -335.427,E2 -335.427} C_VEL
LIN {X 0,Y 608.454,Z 257.32,A -85,B 0,C 180,E1 -338.308,E2 -338.308} C_VEL
LIN {X 0,Y 608.411,Z 257.318,A -85,B 0,C 180,E1 -341.3,E2 -341.3} C_VEL
LIN {X 0,Y 608.421,Z 257.319,A -85,B 0,C 180,E1 -343.905,E2 -343.905} C_VEL
LIN {X 0,Y 608.445,Z 257.319,A -85,B 0,C 180,E1 -346.643,E2 -346.643} C_VEL
LIN {X 0,Y 608.412,Z 257.317,A -85,B 0,C 180,E1 -349.349,E2 -349.349} C_VEL
LIN {X 0,Y 608.434,Z 257.32,A -85,B 0,C 180,E1 -352.032,E2 -352.032} C_VEL
LIN {X 0,Y 608.45,Z 257.316,A -85,B 0,C 180,E1 -354.698,E2 -354.698} C_VEL
LIN {X 0,Y 608.43,Z 257.315,A -85,B 0,C 180,E1 -357.352,E2 -357.352} C_VEL
LIN {X 0,Y 608.464,Z 257.318,A -85,B 0,C 180,E1 -360,E2 -360} C_VEL
LIN {X 0,Y 608.471,Z 257.313,A -85,B 0,C 180,E1 -362.648,E2 -362.648} C_VEL
LIN {X 0,Y 608.422,Z 257.316,A -85,B 0,C 180,E1 -365.302,E2 -365.302} C_VEL
LIN {X 0,Y 608.466,Z 257.319,A -85,B 0,C 180,E1 -367.967,E2 -367.967} C_VEL
LIN {X 0,Y 608.421,Z 257.316,A -85,B 0,C 180,E1 -370.933,E2 -370.933} C_VEL
LIN {X 0,Y 608.43,Z 257.316,A -85,B 0,C 180,E1 -373.357,E2 -373.357} C_VEL
LIN {X 0,Y 608.459,Z 257.321,A -85,B 0,C 180,E1 -376.094,E2 -376.094} C_VEL
LIN {X 0,Y 608.441,Z 257.314,A -85,B 0,C 180,E1 -378.87,E2 -378.87} C_VEL
LIN {X 0,Y 608.453,Z 257.319,A -85,B 0,C 180,E1 -381.692,E2 -381.692} C_VEL
LIN {X 0,Y 608.443,Z 257.314,A -85,B 0,C 180,E1 -384.571,E2 -384.571} C_VEL
LIN {X 0,Y 608.428,Z 257.317,A -85,B 0,C 180,E1 -387.198,E2 -387.198} C_VEL
LIN {X 0,Y 608.477,Z 257.317,A -85,B 0,C 180,E1 -389.973,E2 -389.973} C_VEL
LIN {X 0,Y 608.442,Z 257.314,A -85,B 0,C 180,E1 -392.88,E2 -392.88} C_VEL
LIN {X 0,Y 608.432,Z 257.318,A -85,B 0,C 180,E1 -395.278,E2 -395.278} C_VEL
LIN {X 0,Y 608.468,Z 257.313,A -85,B 0,C 180,E1 -398.241,E2 -398.241} C_VEL
LIN {X 0,Y 608.444,Z 257.318,A -85,B 0,C 180,E1 -401.341,E2 -401.341} C_VEL
LIN {X 0,Y 608.46,Z 257.313,A -85,B 0,C 180,E1 -404.264,E2 -404.264} C_VEL
LIN {X 0,Y 608.429,Z 257.317,A -85,B 0,C 180,E1 -407.038,E2 -407.038} C_VEL
LIN {X 0,Y 608.452,Z 257.321,A -85,B 0,C 180,E1 -409.697,E2 -409.697} C_VEL
LIN {X 0,Y 608.465,Z 257.312,A -85,B 0,C 180,E1 -412.254,E2 -412.254} C_VEL
LIN {X 0,Y 608.436,Z 257.315,A -85,B 0,C 180,E1 -414.722,E2 -414.722} C_VEL
LIN {X 0,Y 608.465,Z 257.322,A -85,B 0,C 180,E1 -417.477,E2 -417.477} C_VEL
LIN {X 0,Y 608.48,Z 257.31,A -85,B 0,C 180,E1 -420.221,E2 -420.221} C_VEL
LIN {X 0,Y 608.463,Z 257.313,A -85,B 0,C 180,E1 -422.795,E2 -422.795} C_VEL
LIN {X 0,Y 608.475,Z 257.451,A -85,B 0,C 180,E1 -424.342,E2 -424.342} C_VEL
LIN {X 0,Y 608.685,Z 269.358,A -85,B 0,C 180,E1 -425.713,E2 -425.713} C_VEL
LIN {X 0,Y 608.624,Z 294.084,A -85,B 0,C 180,E1 -428.492,E2 -428.492} C_VEL
LIN {X 0,Y 608.557,Z 318.021,A -85,B 0,C 180,E1 -431.134,E2 -431.134} C_VEL
LIN {X 0,Y 608.606,Z 322.022,A -85,B 0,C 180,E1 -431.548,E2 -431.548} C_VEL
LIN {X 0,Y 608.697,Z 463.94,A -85,B 0,C 180,E1 -433.272,E2 -433.272} C_VEL
LIN {X 0,Y 608.675,Z 489.91,A -85,B 0,C 180,E1 -433.614,E2 -433.614} C_VEL
LIN {X 0,Y 608.642,Z 505.259,A -85,B 0,C 180,E1 -433.954,E2 -433.954} C_VEL
LIN {X 0,Y 608.606,Z 520.192,A -85,B 0,C 180,E1 -434.426,E2 -434.426} C_VEL
LIN {X 0,Y 608.592,Z 534.619,A -85,B 0,C 180,E1 -435.026,E2 -435.026} C_VEL
LIN {X 0,Y 608.565,Z 547.794,A -85,B 0,C 180,E1 -435.71,E2 -435.71} C_VEL
LIN {X 0,Y 608.548,Z 561.204,A -85,B 0,C 180,E1 -436.561,E2 -436.561} C_VEL
LIN {X 0,Y 608.504,Z 573.392,A -85,B 0,C 180,E1 -437.493,E2 -437.493} C_VEL
LIN {X 0,Y 608.496,Z 584.512,A -85,B 0,C 180,E1 -438.508,E2 -438.508} C_VEL
LIN {X 0,Y 608.476,Z 595.301,A -85,B 0,C 180,E1 -439.687,E2 -439.687} C_VEL
LIN {X 0,Y 608.469,Z 604.292,A -85,B 0,C 180,E1 -440.862,E2 -440.862} C_VEL
LIN {X 0,Y 608.456,Z 611.754,A -85,B 0,C 180,E1 -442.033,E2 -442.033} C_VEL
LIN {X 0,Y 608.44,Z 618.862,A -85,B 0,C 180,E1 -443.4,E2 -443.4} C_VEL
LIN {X 0,Y 608.437,Z 624.162,A -85,B 0,C 180,E1 -444.698,E2 -444.698} C_VEL
LIN {X 0,Y 608.428,Z 628.288,A -85,B 0,C 180,E1 -446.026,E2 -446.026} C_VEL
LIN {X 0,Y 608.424,Z 631.185,A -85,B 0,C 180,E1 -447.352,E2 -447.352} C_VEL
LIN {X 0,Y 608.445,Z 632.912,A -85,B 0,C 180,E1 -448.677,E2 -448.677} C_VEL
LIN {X 0,Y 608.431,Z 633.5,A -85,B 0,C 180,E1 -450,E2 -450} C_VEL
LIN {X 0,Y 608.445,Z 632.912,A -85,B 0,C 180,E1 -451.324,E2 -451.324} C_VEL
LIN {X 0,Y 608.424,Z 631.184,A -85,B 0,C 180,E1 -452.649,E2 -452.649} C_VEL
LIN {X 0,Y 608.428,Z 628.287,A -85,B 0,C 180,E1 -453.974,E2 -453.974} C_VEL
LIN {X 0,Y 608.437,Z 624.16,A -85,B 0,C 180,E1 -455.302,E2 -455.302} C_VEL
LIN {X 0,Y 608.437,Z 618.702,A -85,B 0,C 180,E1 -456.633,E2 -456.633} C_VEL
LIN {X 0,Y 608.456,Z 611.75,A -85,B 0,C 180,E1 -457.968,E2 -457.968} C_VEL
LIN {X 0,Y 608.469,Z 604.288,A -85,B 0,C 180,E1 -459.139,E2 -459.139} C_VEL
LIN {X 0,Y 608.476,Z 595.296,A -85,B 0,C 180,E1 -460.313,E2 -460.313} C_VEL
LIN {X 0,Y 608.497,Z 584.505,A -85,B 0,C 180,E1 -461.493,E2 -461.493} C_VEL
LIN {X 0,Y 608.504,Z 573.384,A -85,B 0,C 180,E1 -462.507,E2 -462.507} C_VEL
LIN {X 0,Y 608.548,Z 561.195,A -85,B 0,C 180,E1 -463.44,E2 -463.44} C_VEL
LIN {X 0,Y 608.573,Z 548.214,A -85,B 0,C 180,E1 -464.266,E2 -464.266} C_VEL
LIN {X 0,Y 608.592,Z 534.605,A -85,B 0,C 180,E1 -464.975,E2 -464.975} C_VEL
LIN {X 0,Y 608.609,Z 520.174,A -85,B 0,C 180,E1 -465.574,E2 -465.574} C_VEL
LIN {X 0,Y 608.644,Z 505.238,A -85,B 0,C 180,E1 -466.046,E2 -466.046} C_VEL
LIN {X 0,Y 608.675,Z 489.895,A -85,B 0,C 180,E1 -466.387,E2 -466.387} C_VEL
LIN {X 0,Y 608.681,Z 461.747,A -85,B 0,C 180,E1 -466.755,E2 -466.755} C_VEL
LIN {X 0,Y 608.692,Z 322.513,A -85,B 0,C 180,E1 -468.443,E2 -468.443} C_VEL
LIN {X 0,Y 608.565,Z 321.416,A -85,B 0,C 180,E1 -468.494,E2 -468.494} C_VEL
LIN {X 0,Y 608.587,Z 297.27,A -85,B 0,C 180,E1 -471.154,E2 -471.154} C_VEL
LIN {X 0,Y 608.666,Z 273.333,A -85,B 0,C 180,E1 -473.837,E2 -473.837} C_VEL
LIN {X 0,Y 608.601,Z 258.035,A -85,B 0,C 180,E1 -475.585,E2 -475.585} C_VEL
LIN {X 0,Y 608.466,Z 257.313,A -85,B 0,C 180,E1 -475.699,E2 -475.699} C_VEL
LIN {X 0,Y 608.474,Z 257.321,A -85,B 0,C 180,E1 -478.62,E2 -478.62} C_VEL
LIN {X 0,Y 608.443,Z 257.314,A -85,B 0,C 180,E1 -481.318,E2 -481.318} C_VEL
LIN {X 0,Y 608.448,Z 257.313,A -85,B 0,C 180,E1 -483.731,E2 -483.731} C_VEL
LIN {X 0,Y 608.463,Z 257.315,A -85,B 0,C 180,E1 -486.092,E2 -486.092} C_VEL
LIN {X 0,Y 608.459,Z 257.32,A -85,B 0,C 180,E1 -488.589,E2 -488.589} C_VEL
LIN {X 0,Y 608.444,Z 257.313,A -85,B 0,C 180,E1 -491.34,E2 -491.34} C_VEL
LIN {X 0,Y 608.455,Z 257.32,A -85,B 0,C 180,E1 -494.264,E2 -494.264} C_VEL
LIN {X 0,Y 608.429,Z 257.316,A -85,B 0,C 180,E1 -497.038,E2 -497.038} C_VEL
LIN {X 0,Y 608.456,Z 257.313,A -85,B 0,C 180,E1 -499.697,E2 -499.697} C_VEL
LIN {X 0,Y 608.465,Z 257.321,A -85,B 0,C 180,E1 -502.254,E2 -502.254} C_VEL
LIN {X 0,Y 608.427,Z 257.316,A -85,B 0,C 180,E1 -505.098,E2 -505.098} C_VEL
LIN {X 0,Y 608.46,Z 257.312,A -85,B 0,C 180,E1 -507.479,E2 -507.479} C_VEL
LIN {X 0,Y 608.481,Z 257.32,A -85,B 0,C 180,E1 -510.221,E2 -510.221} C_VEL
LIN {X 0,Y 608.431,Z 257.316,A -85,B 0,C 180,E1 -512.803,E2 -512.803} C_VEL
LIN {X 0,Y 608.445,Z 257.314,A -85,B 0,C 180,E1 -515.429,E2 -515.429} C_VEL
LIN {X 0,Y 608.455,Z 257.319,A -85,B 0,C 180,E1 -518.308,E2 -518.308} C_VEL
LIN {X 0,Y 608.444,Z 257.313,A -85,B 0,C 180,E1 -521.13,E2 -521.13} C_VEL
LIN {X 0,Y 608.461,Z 257.32,A -85,B 0,C 180,E1 -523.906,E2 -523.906} C_VEL
LIN {X 0,Y 608.434,Z 257.316,A -85,B 0,C 180,E1 -526.643,E2 -526.643} C_VEL
LIN {X 0,Y 608.455,Z 257.313,A -85,B 0,C 180,E1 -529.35,E2 -529.35} C_VEL
LIN {X 0,Y 608.471,Z 257.319,A -85,B 0,C 180,E1 -532.033,E2 -532.033} C_VEL
LIN {X 0,Y 608.425,Z 257.316,A -85,B 0,C 180,E1 -534.698,E2 -534.698} C_VEL
LIN {X 0,Y 608.472,Z 257.312,A -85,B 0,C 180,E1 -537.352,E2 -537.352} C_VEL
LIN {X 0,Y 608.47,Z 257.318,A -85,B 0,C 180,E1 -540,E2 -540} C_VEL
LIN {X 0,Y 608.433,Z 257.315,A -85,B 0,C 180,E1 -542.648,E2 -542.648} C_VEL
LIN {X 0,Y 608.451,Z 257.316,A -85,B 0,C 180,E1 -545.302,E2 -545.302} C_VEL
LIN {X 0,Y 608.438,Z 257.321,A -85,B 0,C 180,E1 -547.968,E2 -547.968} C_VEL
LIN {X 0,Y 608.444,Z 257.317,A -85,B 0,C 180,E1 -549.411,E2 -549.411} C_VEL
LIN {X 0,Y 607.767,Z 257.404,A -85,B 0,C 180,E1 -549.964,E2 -549.964} C_VEL
LIN {X 0,Y 604.921,Z 257.758,A -85,B 0,C 180,E1 -550.86,E2 -550.86} C_VEL
LIN {X 0,Y 602.516,Z 258.06,A -85,B 0,C 180,E1 -551.582,E2 -551.582} C_VEL
LIN {X 0,Y 601.469,Z 258.186,A -85,B 0,C 180,E1 -552.138,E2 -552.138} C_VEL
LIN {X 0,Y 601.377,Z 258.195,A -85,B 0,C 180,E1 -552.326,E2 -552.326} C_VEL
LIN {X 0,Y 601.383,Z 258.193,A -85,B 0,C 180,E1 -554.898,E2 -554.898} C_VEL
LIN {X 0,Y 601.377,Z 258.203,A -85,B 0,C 180,E1 -557.689,E2 -557.689} C_VEL
LIN {X 0,Y 601.383,Z 258.2,A -85,B 0,C 180,E1 -559.81,E2 -559.81} C_VEL
LIN {X 0,Y 601.378,Z 258.197,A -85,B 0,C 180,E1 -561.961,E2 -561.961} C_VEL
LIN {X 0,Y 601.376,Z 258.195,A -85,B 0,C 180,E1 -564.88,E2 -564.88} C_VEL
LIN {X 0,Y 601.399,Z 258.199,A -85,B 0,C 180,E1 -567.358,E2 -567.358} C_VEL
LIN {X 0,Y 601.374,Z 258.195,A -85,B 0,C 180,E1 -570.167,E2 -570.167} C_VEL
LIN {X 0,Y 601.383,Z 258.194,A -85,B 0,C 180,E1 -572.709,E2 -572.709} C_VEL
LIN {X 0,Y 601.365,Z 258.201,A -85,B 0,C 180,E1 -575.107,E2 -575.107} C_VEL
LIN {X 0,Y 601.4,Z 258.201,A -85,B 0,C 180,E1 -577.422,E2 -577.422} C_VEL
LIN {X 0,Y 601.357,Z 258.198,A -85,B 0,C 180,E1 -579.999,E2 -579.999} C_VEL
LIN {X 0,Y 601.353,Z 258.198,A -85,B 0,C 180,E1 -582.676,E2 -582.676} C_VEL
LIN {X 0,Y 601.367,Z 258.195,A -85,B 0,C 180,E1 -584.529,E2 -584.529} C_VEL
LIN {X 0,Y 601.362,Z 258.203,A -85,B 0,C 180,E1 -587.415,E2 -587.415} C_VEL
LIN {X 0,Y 601.379,Z 258.194,A -85,B 0,C 180,E1 -590.472,E2 -590.472} C_VEL
LIN {X 0,Y 601.375,Z 258.201,A -85,B 0,C 180,E1 -593.415,E2 -593.415} C_VEL
LIN {X 0,Y 601.371,Z 258.194,A -85,B 0,C 180,E1 -596.073,E2 -596.073} C_VEL
LIN {X 0,Y 601.385,Z 258.195,A -85,B 0,C 180,E1 -598.551,E2 -598.551} C_VEL
LIN {X 0,Y 601.406,Z 258.196,A -85,B 0,C 180,E1 -601.371,E2 -601.371} C_VEL
LIN {X 0,Y 601.353,Z 258.197,A -85,B 0,C 180,E1 -604.145,E2 -604.145} C_VEL
LIN {X 0,Y 601.363,Z 258.2,A -85,B 0,C 180,E1 -606.587,E2 -606.587} C_VEL
LIN {X 0,Y 601.355,Z 258.235,A -85,B 0,C 180,E1 -607.994,E2 -607.994} C_VEL
LIN {X 0,Y 601.666,Z 263.81,A -85,B 0,C 180,E1 -608.77,E2 -608.77} C_VEL
LIN {X 0,Y 601.58,Z 283.225,A -85,B 0,C 180,E1 -611.384,E2 -611.384} C_VEL
LIN {X 0,Y 602.006,Z 286.339,A -85,B 0,C 180,E1 -611.437,E2 -611.437} C_VEL
LIN {X 0,Y 601.881,Z 447.964,A -85,B 0,C 180,E1 -613.432,E2 -613.432} C_VEL
LIN {X 0,Y 601.824,Z 463.646,A -85,B 0,C 180,E1 -613.767,E2 -613.767} C_VEL
LIN {X 0,Y 601.753,Z 478.998,A -85,B 0,C 180,E1 -614.244,E2 -614.244} C_VEL
LIN {X 0,Y 601.725,Z 493.677,A -85,B 0,C 180,E1 -614.85,E2 -614.85} C_VEL
LIN {X 0,Y 601.659,Z 506.976,A -85,B 0,C 180,E1 -615.541,E2 -615.541} C_VEL
LIN {X 0,Y 601.604,Z 519.798,A -85,B 0,C 180,E1 -616.351,E2 -616.351} C_VEL
LIN {X 0,Y 601.541,Z 531.785,A -85,B 0,C 180,E1 -617.26,E2 -617.26} C_VEL
LIN {X 0,Y 601.489,Z 542.277,A -85,B 0,C 180,E1 -618.201,E2 -618.201} C_VEL
LIN {X 0,Y 601.43,Z 551.992,A -85,B 0,C 180,E1 -619.224,E2 -619.224} C_VEL
LIN {X 0,Y 601.428,Z 561.524,A -85,B 0,C 180,E1 -620.414,E2 -620.414} C_VEL
LIN {X 0,Y 601.378,Z 569.458,A -85,B 0,C 180,E1 -621.6,E2 -621.6} C_VEL
LIN {X 0,Y 601.368,Z 576.87,A -85,B 0,C 180,E1 -622.951,E2 -622.951} C_VEL
LIN {X 0,Y 601.372,Z 582.758,A -85,B 0,C 180,E1 -624.299,E2 -624.299} C_VEL
LIN {X 0,Y 601.329,Z 586.24,A -85,B 0,C 180,E1 -625.307,E2 -625.307} C_VEL
LIN {X 0,Y 601.336,Z 589.789,A -85,B 0,C 180,E1 -626.65,E2 -626.65} C_VEL
LIN {X 0,Y 601.343,Z 592.139,A -85,B 0,C 180,E1 -627.99,E2 -627.99} C_VEL
LIN {X 0,Y 601.334,Z 593.337,A -85,B 0,C 180,E1 -629.33,E2 -629.33} C_VEL
LIN {X 0,Y 601.335,Z 593.361,A -85,B 0,C 180,E1 -630.669,E2 -630.669} C_VEL
LIN {X 0,Y 601.343,Z 592.245,A -85,B 0,C 180,E1 -632.009,E2 -632.009} C_VEL
LIN {X 0,Y 601.339,Z 589.983,A -85,B 0,C 180,E1 -633.35,E2 -633.35} C_VEL
LIN {X 0,Y 601.329,Z 586.526,A -85,B 0,C 180,E1 -634.692,E2 -634.692} C_VEL
LIN {X 0,Y 601.357,Z 581.799,A -85,B 0,C 180,E1 -636.037,E2 -636.037} C_VEL
LIN {X 0,Y 601.364,Z 575.668,A -85,B 0,C 180,E1 -637.386,E2 -637.386} C_VEL
LIN {X 0,Y 601.387,Z 567.952,A -85,B 0,C 180,E1 -638.738,E2 -638.738} C_VEL
LIN {X 0,Y 601.428,Z 559.709,A -85,B 0,C 180,E1 -639.925,E2 -639.925} C_VEL
LIN {X 0,Y 601.443,Z 549.366,A -85,B 0,C 180,E1 -641.164,E2 -641.164} C_VEL
LIN {X 0,Y 601.503,Z 537.788,A -85,B 0,C 180,E1 -642.312,E2 -642.312} C_VEL
LIN {X 0,Y 601.557,Z 526.467,A -85,B 0,C 180,E1 -643.254,E2 -643.254} C_VEL
LIN {X 0,Y 601.623,Z 513.318,A -85,B 0,C 180,E1 -644.167,E2 -644.167} C_VEL
LIN {X 0,Y 601.661,Z 500.764,A -85,B 0,C 180,E1 -644.891,E2 -644.891} C_VEL
LIN {X 0,Y 601.757,Z 485.841,A -85,B 0,C 180,E1 -645.582,E2 -645.582} C_VEL
LIN {X 0,Y 601.807,Z 471.353,A -85,B 0,C 180,E1 -646.102,E2 -646.102} C_VEL
LIN {X 0,Y 601.874,Z 456.057,A -85,B 0,C 180,E1 -646.503,E2 -646.503} C_VEL
LIN {X 0,Y 601.894,Z 440.192,A -85,B 0,C 180,E1 -646.77,E2 -646.77} C_VEL
LIN {X 0,Y 601.904,Z 284.825,A -85,B 0,C 180,E1 -648.675,E2 -648.675} C_VEL
LIN {X 0,Y 601.58,Z 282.965,A -85,B 0,C 180,E1 -648.729,E2 -648.729} C_VEL
LIN {X 0,Y 601.636,Z 261.844,A -85,B 0,C 180,E1 -651.59,E2 -651.59} C_VEL
LIN {X 0,Y 601.381,Z 258.197,A -85,B 0,C 180,E1 -652.113,E2 -652.113} C_VEL
LIN {X 0,Y 601.385,Z 258.201,A -85,B 0,C 180,E1 -654.879,E2 -654.879} C_VEL
LIN {X 0,Y 601.391,Z 258.197,A -85,B 0,C 180,E1 -657.358,E2 -657.358} C_VEL
LIN {X 0,Y 601.369,Z 258.199,A -85,B 0,C 180,E1 -659.396,E2 -659.396} C_VEL
LIN {X 0,Y 601.376,Z 258.195,A -85,B 0,C 180,E1 -661.728,E2 -661.728} C_VEL
LIN {X 0,Y 601.38,Z 258.194,A -85,B 0,C 180,E1 -664.121,E2 -664.121} C_VEL
LIN {X 0,Y 601.384,Z 258.198,A -85,B 0,C 180,E1 -666.584,E2 -666.584} C_VEL
LIN {X 0,Y 601.383,Z 258.194,A -85,B 0,C 180,E1 -669.529,E2 -669.529} C_VEL
LIN {X 0,Y 601.369,Z 258.195,A -85,B 0,C 180,E1 -671.77,E2 -671.77} C_VEL
LIN {X 0,Y 601.397,Z 258.197,A -85,B 0,C 180,E1 -674.532,E2 -674.532} C_VEL
LIN {X 0,Y 601.353,Z 258.198,A -85,B 0,C 180,E1 -677.324,E2 -677.324} C_VEL
LIN {X 0,Y 601.356,Z 258.197,A -85,B 0,C 180,E1 -679.433,E2 -679.433} C_VEL
LIN {X 0,Y 601.336,Z 258.199,A -85,B 0,C 180,E1 -681.726,E2 -681.726} C_VEL
LIN {X 0,Y 601.343,Z 258.2,A -85,B 0,C 180,E1 -684.242,E2 -684.242} C_VEL
LIN {X 0,Y 601.405,Z 258.2,A -85,B 0,C 180,E1 -686.685,E2 -686.685} C_VEL
LIN {X 0,Y 601.383,Z 258.196,A -85,B 0,C 180,E1 -689.056,E2 -689.056} C_VEL
LIN {X 0,Y 601.379,Z 258.194,A -85,B 0,C 180,E1 -691.37,E2 -691.37} C_VEL
LIN {X 0,Y 601.365,Z 258.195,A -85,B 0,C 180,E1 -693.634,E2 -693.634} C_VEL
LIN {X 0,Y 601.388,Z 258.194,A -85,B 0,C 180,E1 -695.857,E2 -695.857} C_VEL
LIN {X 0,Y 601.39,Z 258.198,A -85,B 0,C 180,E1 -698.76,E2 -698.76} C_VEL
LIN {X 0,Y 601.357,Z 258.196,A -85,B 0,C 180,E1 -701.606,E2 -701.606} C_VEL
LIN {X 0,Y 601.393,Z 258.203,A -85,B 0,C 180,E1 -704.408,E2 -704.408} C_VEL
LIN {X 0,Y 601.361,Z 258.196,A -85,B 0,C 180,E1 -707.17,E2 -707.17} C_VEL
LIN {X 0,Y 601.374,Z 258.194,A -85,B 0,C 180,E1 -709.223,E2 -709.223} C_VEL
LIN {X 0,Y 601.402,Z 258.195,A -85,B 0,C 180,E1 -711.939,E2 -711.939} C_VEL
LIN {X 0,Y 601.414,Z 258.193,A -85,B 0,C 180,E1 -714.636,E2 -714.636} C_VEL
LIN {X 0,Y 601.4,Z 258.191,A -85,B 0,C 180,E1 -717.321,E2 -717.321} C_VEL
LIN {X 0,Y 601.433,Z 258.194,A -85,B 0,C 180,E1 -720,E2 -720} C_VEL
LIN {X 0,Y 601.433,Z 258.189,A -85,B 0,C 180,E1 -722.679,E2 -722.679} C_VEL
LIN {X 0,Y 601.39,Z 258.192,A -85,B 0,C 180,E1 -725.364,E2 -725.364} C_VEL
LIN {X 0,Y 601.431,Z 258.197,A -85,B 0,C 180,E1 -728.061,E2 -728.061} C_VEL
LIN {X 0,Y 601.399,Z 258.191,A -85,B 0,C 180,E1 -730.999,E2 -730.999} C_VEL
LIN {X 0,Y 601.394,Z 258.194,A -85,B 0,C 180,E1 -733.516,E2 -733.516} C_VEL
LIN {X 0,Y 601.439,Z 258.192,A -85,B 0,C 180,E1 -736.287,E2 -736.287} C_VEL
LIN {X 0,Y 601.406,Z 258.19,A -85,B 0,C 180,E1 -739.099,E2 -739.099} C_VEL
LIN {X 0,Y 601.391,Z 258.193,A -85,B 0,C 180,E1 -741.24,E2 -741.24} C_VEL
LIN {X 0,Y 601.462,Z 258.188,A -85,B 0,C 180,E1 -744.14,E2 -744.14} C_VEL
LIN {X 0,Y 601.39,Z 258.192,A -85,B 0,C 180,E1 -747.114,E2 -747.114} C_VEL
LIN {X 0,Y 601.403,Z 258.194,A -85,B 0,C 180,E1 -749.394,E2 -749.394} C_VEL
LIN {X 0,Y 601.4,Z 258.2,A -85,B 0,C 180,E1 -751.727,E2 -751.727} C_VEL
LIN {X 0,Y 601.423,Z 258.193,A -85,B 0,C 180,E1 -754.119,E2 -754.119} C_VEL
LIN {X 0,Y 601.396,Z 258.191,A -85,B 0,C 180,E1 -756.583,E2 -756.583} C_VEL
LIN {X 0,Y 601.395,Z 258.193,A -85,B 0,C 180,E1 -759.128,E2 -759.128} C_VEL
LIN {X 0,Y 601.423,Z 258.197,A -85,B 0,C 180,E1 -761.765,E2 -761.765} C_VEL
LIN {X 0,Y 601.396,Z 258.192,A -85,B 0,C 180,E1 -764.533,E2 -764.533} C_VEL
LIN {X 0,Y 601.411,Z 258.197,A -85,B 0,C 180,E1 -767.409,E2 -767.409} C_VEL
LIN {X 0,Y 601.4,Z 258.194,A -85,B 0,C 180,E1 -770.004,E2 -770.004} C_VEL
LIN {X 0,Y 601.43,Z 258.187,A -85,B 0,C 180,E1 -772.619,E2 -772.619} C_VEL
LIN {X 0,Y 601.402,Z 258.195,A -85,B 0,C 180,E1 -775.067,E2 -775.067} C_VEL
LIN {X 0,Y 601.433,Z 258.197,A -85,B 0,C 180,E1 -777.485,E2 -777.485} C_VEL
LIN {X 0,Y 601.429,Z 258.192,A -85,B 0,C 180,E1 -779.851,E2 -779.851} C_VEL
LIN {X 0,Y 601.405,Z 258.192,A -85,B 0,C 180,E1 -782.639,E2 -782.639} C_VEL
LIN {X 0,Y 601.452,Z 258.35,A -85,B 0,C 180,E1 -784.125,E2 -784.125} C_VEL
LIN {X 0,Y 601.882,Z 262.168,A -85,B 0,C 180,E1 -784.589,E2 -784.589} C_VEL
LIN {X 0,Y 601.81,Z 285.855,A -85,B 0,C 180,E1 -787.305,E2 -787.305} C_VEL
LIN {X 0,Y 601.689,Z 313.234,A -85,B 0,C 180,E1 -790.378,E2 -790.378} C_VEL
LIN {X 0,Y 601.633,Z 321.729,A -85,B 0,C 180,E1 -791.319,E2 -791.319} C_VEL
LIN {X 0,Y 602.054,Z 326.022,A -85,B 0,C 180,E1 -791.389,E2 -791.389} C_VEL
LIN {X 0,Y 601.878,Z 488.492,A -85,B 0,C 180,E1 -793.396,E2 -793.396} C_VEL
LIN {X 0,Y 601.815,Z 504.496,A -85,B 0,C 180,E1 -793.746,E2 -793.746} C_VEL
LIN {X 0,Y 601.767,Z 519.055,A -85,B 0,C 180,E1 -794.201,E2 -794.201} C_VEL
LIN {X 0,Y 601.72,Z 532.766,A -85,B 0,C 180,E1 -794.764,E2 -794.764} C_VEL
LIN {X 0,Y 601.662,Z 546.238,A -85,B 0,C 180,E1 -795.455,E2 -795.455} C_VEL
LIN {X 0,Y 601.617,Z 559.452,A -85,B 0,C 180,E1 -796.283,E2 -796.283} C_VEL
LIN {X 0,Y 601.532,Z 571.288,A -85,B 0,C 180,E1 -797.175,E2 -797.175} C_VEL
LIN {X 0,Y 601.488,Z 582.751,A -85,B 0,C 180,E1 -798.201,E2 -798.201} C_VEL
LIN {X 0,Y 601.431,Z 592.391,A -85,B 0,C 180,E1 -799.224,E2 -799.224} C_VEL
LIN {X 0,Y 601.428,Z 601.857,A -85,B 0,C 180,E1 -800.415,E2 -800.415} C_VEL
LIN {X 0,Y 601.368,Z 609.732,A -85,B 0,C 180,E1 -801.6,E2 -801.6} C_VEL
LIN {X 0,Y 601.368,Z 617.089,A -85,B 0,C 180,E1 -802.952,E2 -802.952} C_VEL
LIN {X 0,Y 601.371,Z 622.925,A -85,B 0,C 180,E1 -804.299,E2 -804.299} C_VEL
LIN {X 0,Y 601.33,Z 626.384,A -85,B 0,C 180,E1 -805.308,E2 -805.308} C_VEL
LIN {X 0,Y 601.337,Z 629.887,A -85,B 0,C 180,E1 -806.65,E2 -806.65} C_VEL
LIN {X 0,Y 601.341,Z 632.192,A -85,B 0,C 180,E1 -807.991,E2 -807.991} C_VEL
LIN {X 0,Y 601.337,Z 633.35,A -85,B 0,C 180,E1 -809.331,E2 -809.331} C_VEL
LIN {X 0,Y 601.337,Z 633.35,A -85,B 0,C 180,E1 -810.67,E2 -810.67} C_VEL
LIN {X 0,Y 601.341,Z 632.191,A -85,B 0,C 180,E1 -812.01,E2 -812.01} C_VEL
LIN {X 0,Y 601.337,Z 629.885,A -85,B 0,C 180,E1 -813.35,E2 -813.35} C_VEL
LIN {X 0,Y 601.33,Z 626.382,A -85,B 0,C 180,E1 -814.693,E2 -814.693} C_VEL
LIN {X 0,Y 601.352,Z 621.606,A -85,B 0,C 180,E1 -816.038,E2 -816.038} C_VEL
LIN {X 0,Y 601.366,Z 615.423,A -85,B 0,C 180,E1 -817.386,E2 -817.386} C_VEL
LIN {X 0,Y 601.387,Z 607.651,A -85,B 0,C 180,E1 -818.739,E2 -818.739} C_VEL
LIN {X 0,Y 601.427,Z 599.367,A -85,B 0,C 180,E1 -819.926,E2 -819.926} C_VEL
LIN {X 0,Y 601.461,Z 588.928,A -85,B 0,C 180,E1 -821.165,E2 -821.165} C_VEL
LIN {X 0,Y 601.514,Z 579.188,A -85,B 0,C 180,E1 -822.141,E2 -822.141} C_VEL
LIN {X 0,Y 601.57,Z 567.011,A -85,B 0,C 180,E1 -823.169,E2 -823.169} C_VEL
LIN {X 0,Y 601.607,Z 555.071,A -85,B 0,C 180,E1 -824.012,E2 -824.012} C_VEL
LIN {X 0,Y 601.669,Z 541.519,A -85,B 0,C 180,E1 -824.805,E2 -824.805} C_VEL
LIN {X 0,Y 601.765,Z 526.833,A -85,B 0,C 180,E1 -825.496,E2 -825.496} C_VEL
LIN {X 0,Y 601.788,Z 512.606,A -85,B 0,C 180,E1 -826.016,E2 -826.016} C_VEL
LIN {X 0,Y 601.86,Z 497.658,A -85,B 0,C 180,E1 -826.421,E2 -826.421} C_VEL
LIN {X 0,Y 601.87,Z 482.658,A -85,B 0,C 180,E1 -826.69,E2 -826.69} C_VEL
LIN {X 0,Y 601.991,Z 323.572,A -85,B 0,C 180,E1 -828.643,E2 -828.643} C_VEL
LIN {X 0,Y 601.653,Z 321.599,A -85,B 0,C 180,E1 -828.694,E2 -828.694} C_VEL
LIN {X 0,Y 601.755,Z 295.674,A -85,B 0,C 180,E1 -831.586,E2 -831.586} C_VEL
LIN {X 0,Y 601.877,Z 271.05,A -85,B 0,C 180,E1 -834.385,E2 -834.385} C_VEL
LIN {X 0,Y 601.864,Z 260.566,A -85,B 0,C 180,E1 -835.598,E2 -835.598} C_VEL
LIN {X 0,Y 601.412,Z 258.195,A -85,B 0,C 180,E1 -835.909,E2 -835.909} C_VEL
LIN {X 0,Y 601.431,Z 258.198,A -85,B 0,C 180,E1 -838.627,E2 -838.627} C_VEL
LIN {X 0,Y 601.419,Z 258.189,A -85,B 0,C 180,E1 -841.454,E2 -841.454} C_VEL
LIN {X 0,Y 601.421,Z 258.192,A -85,B 0,C 180,E1 -844.119,E2 -844.119} C_VEL
LIN {X 0,Y 601.399,Z 258.2,A -85,B 0,C 180,E1 -846.584,E2 -846.584} C_VEL
LIN {X 0,Y 601.404,Z 258.191,A -85,B 0,C 180,E1 -849.128,E2 -849.128} C_VEL
LIN {X 0,Y 601.423,Z 258.189,A -85,B 0,C 180,E1 -851.766,E2 -851.766} C_VEL
LIN {X 0,Y 601.4,Z 258.199,A -85,B 0,C 180,E1 -854.533,E2 -854.533} C_VEL
LIN {X 0,Y 601.411,Z 258.189,A -85,B 0,C 180,E1 -857.41,E2 -857.41} C_VEL
LIN {X 0,Y 601.403,Z 258.195,A -85,B 0,C 180,E1 -860.004,E2 -860.004} C_VEL
LIN {X 0,Y 601.432,Z 258.192,A -85,B 0,C 180,E1 -862.619,E2 -862.619} C_VEL
LIN {X 0,Y 601.391,Z 258.192,A -85,B 0,C 180,E1 -865.067,E2 -865.067} C_VEL
LIN {X 0,Y 601.429,Z 258.188,A -85,B 0,C 180,E1 -867.484,E2 -867.484} C_VEL
LIN {X 0,Y 601.434,Z 258.191,A -85,B 0,C 180,E1 -869.852,E2 -869.852} C_VEL
LIN {X 0,Y 601.387,Z 258.195,A -85,B 0,C 180,E1 -872.644,E2 -872.644} C_VEL
LIN {X 0,Y 601.389,Z 258.192,A -85,B 0,C 180,E1 -875.121,E2 -875.121} C_VEL
LIN {X 0,Y 601.42,Z 258.189,A -85,B 0,C 180,E1 -877.395,E2 -877.395} C_VEL
LIN {X 0,Y 601.396,Z 258.2,A -85,B 0,C 180,E1 -880.19,E2 -880.19} C_VEL
LIN {X 0,Y 601.406,Z 258.19,A -85,B 0,C 180,E1 -883.013,E2 -883.013} C_VEL
LIN {X 0,Y 601.427,Z 258.196,A -85,B 0,C 180,E1 -885.909,E2 -885.909} C_VEL
LIN {X 0,Y 601.405,Z 258.192,A -85,B 0,C 180,E1 -888.541,E2 -888.541} C_VEL
LIN {X 0,Y 601.405,Z 258.191,A -85,B 0,C 180,E1 -891.262,E2 -891.262} C_VEL
LIN {X 0,Y 601.404,Z 258.2,A -85,B 0,C 180,E1 -893.963,E2 -893.963} C_VEL
LIN {X 0,Y 601.365,Z 258.196,A -85,B 0,C 180,E1 -896.65,E2 -896.65} C_VEL
LIN {X 0,Y 601.441,Z 258.188,A -85,B 0,C 180,E1 -899.331,E2 -899.331} C_VEL
LIN {X 0,Y 601.417,Z 258.196,A -85,B 0,C 180,E1 -902.009,E2 -902.009} C_VEL
LIN {X 0,Y 601.382,Z 258.193,A -85,B 0,C 180,E1 -904.692,E2 -904.692} C_VEL
LIN {X 0,Y 601.403,Z 258.195,A -85,B 0,C 180,E1 -907.386,E2 -907.386} C_VEL
LIN {X 0,Y 601.396,Z 258.195,A -85,B 0,C 180,E1 -910.096,E2 -910.096} C_VEL
LIN {X 0,Y 601.377,Z 258.195,A -85,B 0,C 180,E1 -912.326,E2 -912.326} C_VEL
LIN {X 0,Y 600.692,Z 258.281,A -85,B 0,C 180,E1 -912.886,E2 -912.886} C_VEL
LIN {X 0,Y 597.842,Z 258.642,A -85,B 0,C 180,E1 -913.794,E2 -913.794} C_VEL
LIN {X 0,Y 595.445,Z 258.937,A -85,B 0,C 180,E1 -914.524,E2 -914.524} C_VEL
LIN {X 0,Y 594.416,Z 259.063,A -85,B 0,C 180,E1 -915.087,E2 -915.087} C_VEL
LIN {X 0,Y 594.331,Z 259.074,A -85,B 0,C 180,E1 -915.278,E2 -915.278} C_VEL
LIN {X 0,Y 594.325,Z 259.077,A -85,B 0,C 180,E1 -917.906,E2 -917.906} C_VEL
LIN {X 0,Y 594.373,Z 259.067,A -85,B 0,C 180,E1 -920.777,E2 -920.777} C_VEL
LIN {X 0,Y 594.342,Z 259.078,A -85,B 0,C 180,E1 -923.706,E2 -923.706} C_VEL
LIN {X 0,Y 594.354,Z 259.069,A -85,B 0,C 180,E1 -926.701,E2 -926.701} C_VEL
LIN {X 0,Y 594.337,Z 259.076,A -85,B 0,C 180,E1 -929.779,E2 -929.779} C_VEL
LIN {X 0,Y 594.333,Z 259.072,A -85,B 0,C 180,E1 -932.149,E2 -932.149} C_VEL
LIN {X 0,Y 594.328,Z 259.072,A -85,B 0,C 180,E1 -934.583,E2 -934.583} C_VEL
LIN {X 0,Y 594.355,Z 259.075,A -85,B 0,C 180,E1 -937.603,E2 -937.603} C_VEL
LIN {X 0,Y 594.316,Z 259.074,A -85,B 0,C 180,E1 -940.571,E2 -940.571} C_VEL
LIN {X 0,Y 594.34,Z 259.081,A -85,B 0,C 180,E1 -943.302,E2 -943.302} C_VEL
LIN {X 0,Y 594.314,Z 259.074,A -85,B 0,C 180,E1 -946.166,E2 -946.166} C_VEL
LIN {X 0,Y 594.32,Z 259.074,A -85,B 0,C 180,E1 -948.53,E2 -948.53} C_VEL
LIN {X 0,Y 594.324,Z 259.081,A -85,B 0,C 180,E1 -951.303,E2 -951.303} C_VEL
LIN {X 0,Y 594.311,Z 259.076,A -85,B 0,C 180,E1 -953.752,E2 -953.752} C_VEL
LIN {X 0,Y 594.319,Z 259.073,A -85,B 0,C 180,E1 -956.234,E2 -956.234} C_VEL
LIN {X 0,Y 594.338,Z 259.074,A -85,B 0,C 180,E1 -958.647,E2 -958.647} C_VEL
LIN {X 0,Y 594.344,Z 259.08,A -85,B 0,C 180,E1 -961.049,E2 -961.049} C_VEL
LIN {X 0,Y 594.35,Z 259.076,A -85,B 0,C 180,E1 -963.298,E2 -963.298} C_VEL
LIN {X 0,Y 594.332,Z 259.074,A -85,B 0,C 180,E1 -966.293,E2 -966.293} C_VEL
LIN {X 0,Y 594.353,Z 259.215,A -85,B 0,C 180,E1 -967.857,E2 -967.857} C_VEL
LIN {X 0,Y 594.696,Z 263.814,A -85,B 0,C 180,E1 -968.509,E2 -968.509} C_VEL
LIN {X 0,Y 594.621,Z 283.084,A -85,B 0,C 180,E1 -971.151,E2 -971.151} C_VEL
LIN {X 0,Y 595.275,Z 286.976,A -85,B 0,C 180,E1 -971.226,E2 -971.226} C_VEL
LIN {X 0,Y 595.092,Z 448.418,A -85,B 0,C 180,E1 -973.245,E2 -973.245} C_VEL
LIN {X 0,Y 595.017,Z 463.667,A -85,B 0,C 180,E1 -973.576,E2 -973.576} C_VEL
LIN {X 0,Y 594.911,Z 479.012,A -85,B 0,C 180,E1 -974.058,E2 -974.058} C_VEL
LIN {X 0,Y 594.857,Z 493.687,A -85,B 0,C 180,E1 -974.671,E2 -974.671} C_VEL
LIN {X 0,Y 594.745,Z 506.989,A -85,B 0,C 180,E1 -975.369,E2 -975.369} C_VEL
LIN {X 0,Y 594.67,Z 519.984,A -85,B 0,C 180,E1 -976.201,E2 -976.201} C_VEL
LIN {X 0,Y 594.553,Z 532.853,A -85,B 0,C 180,E1 -977.194,E2 -977.194} C_VEL
LIN {X 0,Y 594.469,Z 544.058,A -85,B 0,C 180,E1 -978.232,E2 -978.232} C_VEL
LIN {X 0,Y 594.412,Z 554.943,A -85,B 0,C 180,E1 -979.44,E2 -979.44} C_VEL
LIN {X 0,Y 594.357,Z 563.988,A -85,B 0,C 180,E1 -980.643,E2 -980.643} C_VEL
LIN {X 0,Y 594.325,Z 571.483,A -85,B 0,C 180,E1 -981.842,E2 -981.842} C_VEL
LIN {X 0,Y 594.277,Z 578.488,A -85,B 0,C 180,E1 -983.208,E2 -983.208} C_VEL
LIN {X 0,Y 594.273,Z 583.997,A -85,B 0,C 180,E1 -984.571,E2 -984.571} C_VEL
LIN {X 0,Y 594.254,Z 588.17,A -85,B 0,C 180,E1 -985.931,E2 -985.931} C_VEL
LIN {X 0,Y 594.221,Z 591.112,A -85,B 0,C 180,E1 -987.288,E2 -987.288} C_VEL
LIN {X 0,Y 594.244,Z 592.88,A -85,B 0,C 180,E1 -988.644,E2 -988.644} C_VEL
LIN {X 0,Y 594.234,Z 593.496,A -85,B 0,C 180,E1 -990,E2 -990} C_VEL
LIN {X 0,Y 594.246,Z 592.944,A -85,B 0,C 180,E1 -991.355,E2 -991.355} C_VEL
LIN {X 0,Y 594.224,Z 591.26,A -85,B 0,C 180,E1 -992.711,E2 -992.711} C_VEL
LIN {X 0,Y 594.254,Z 588.407,A -85,B 0,C 180,E1 -994.069,E2 -994.069} C_VEL
LIN {X 0,Y 594.273,Z 584.326,A -85,B 0,C 180,E1 -995.429,E2 -995.429} C_VEL
LIN {X 0,Y 594.276,Z 578.917,A -85,B 0,C 180,E1 -996.791,E2 -996.791} C_VEL
LIN {X 0,Y 594.324,Z 572.018,A -85,B 0,C 180,E1 -998.158,E2 -998.158} C_VEL
LIN {X 0,Y 594.339,Z 563.416,A -85,B 0,C 180,E1 -999.529,E2 -999.529} C_VEL
LIN {X 0,Y 594.401,Z 554.267,A -85,B 0,C 180,E1 -1000.732,E2 -1000.732} C_VEL
LIN {X 0,Y 594.466,Z 543.213,A -85,B 0,C 180,E1 -1001.94,E2 -1001.94} C_VEL
LIN {X 0,Y 594.56,Z 531.839,A -85,B 0,C 180,E1 -1002.978,E2 -1002.978} C_VEL
LIN {X 0,Y 594.66,Z 519.456,A -85,B 0,C 180,E1 -1003.925,E2 -1003.925} C_VEL
LIN {X 0,Y 594.725,Z 507.047,A -85,B 0,C 180,E1 -1004.718,E2 -1004.718} C_VEL
LIN {X 0,Y 594.853,Z 493.75,A -85,B 0,C 180,E1 -1005.416,E2 -1005.416} C_VEL
LIN {X 0,Y 594.905,Z 479.079,A -85,B 0,C 180,E1 -1006.03,E2 -1006.03} C_VEL
LIN {X 0,Y 595.036,Z 463.937,A -85,B 0,C 180,E1 -1006.506,E2 -1006.506} C_VEL
LIN {X 0,Y 595.084,Z 448.21,A -85,B 0,C 180,E1 -1006.849,E2 -1006.849} C_VEL
LIN {X 0,Y 595.292,Z 286.845,A -85,B 0,C 180,E1 -1008.865,E2 -1008.865} C_VEL
LIN {X 0,Y 594.637,Z 283.065,A -85,B 0,C 180,E1 -1008.942,E2 -1008.942} C_VEL
LIN {X 0,Y 594.733,Z 263.155,A -85,B 0,C 180,E1 -1011.671,E2 -1011.671} C_VEL
LIN {X 0,Y 594.352,Z 259.075,A -85,B 0,C 180,E1 -1012.269,E2 -1012.269} C_VEL
LIN {X 0,Y 594.347,Z 259.078,A -85,B 0,C 180,E1 -1015.194,E2 -1015.194} C_VEL
LIN {X 0,Y 594.342,Z 259.074,A -85,B 0,C 180,E1 -1017.518,E2 -1017.518} C_VEL
LIN {X 0,Y 594.328,Z 259.073,A -85,B 0,C 180,E1 -1019.779,E2 -1019.779} C_VEL
LIN {X 0,Y 594.343,Z 259.071,A -85,B 0,C 180,E1 -1022.148,E2 -1022.148} C_VEL
LIN {X 0,Y 594.364,Z 259.073,A -85,B 0,C 180,E1 -1024.581,E2 -1024.581} C_VEL
LIN {X 0,Y 594.351,Z 259.07,A -85,B 0,C 180,E1 -1027.603,E2 -1027.603} C_VEL
LIN {X 0,Y 594.352,Z 259.075,A -85,B 0,C 180,E1 -1030.568,E2 -1030.568} C_VEL
LIN {X 0,Y 594.335,Z 259.073,A -85,B 0,C 180,E1 -1033.302,E2 -1033.302} C_VEL
LIN {X 0,Y 594.332,Z 259.073,A -85,B 0,C 180,E1 -1036.164,E2 -1036.164} C_VEL
LIN {X 0,Y 594.356,Z 259.074,A -85,B 0,C 180,E1 -1038.534,E2 -1038.534} C_VEL
LIN {X 0,Y 594.317,Z 259.075,A -85,B 0,C 180,E1 -1041.304,E2 -1041.304} C_VEL
LIN {X 0,Y 594.305,Z 259.073,A -85,B 0,C 180,E1 -1043.752,E2 -1043.752} C_VEL
LIN {X 0,Y 594.334,Z 259.075,A -85,B 0,C 180,E1 -1046.236,E2 -1046.236} C_VEL
LIN {X 0,Y 594.339,Z 259.081,A -85,B 0,C 180,E1 -1048.648,E2 -1048.648} C_VEL
LIN {X 0,Y 594.336,Z 259.074,A -85,B 0,C 180,E1 -1051.05,E2 -1051.05} C_VEL
LIN {X 0,Y 594.351,Z 259.07,A -85,B 0,C 180,E1 -1053.299,E2 -1053.299} C_VEL
LIN {X 0,Y 594.329,Z 259.072,A -85,B 0,C 180,E1 -1055.579,E2 -1055.579} C_VEL
LIN {X 0,Y 594.344,Z 259.081,A -85,B 0,C 180,E1 -1058.496,E2 -1058.496} C_VEL
LIN {X 0,Y 594.339,Z 259.07,A -85,B 0,C 180,E1 -1061.381,E2 -1061.381} C_VEL
LIN {X 0,Y 594.337,Z 259.078,A -85,B 0,C 180,E1 -1064.218,E2 -1064.218} C_VEL
LIN {X 0,Y 594.316,Z 259.075,A -85,B 0,C 180,E1 -1067.016,E2 -1067.016} C_VEL
LIN {X 0,Y 594.362,Z 259.068,A -85,B 0,C 180,E1 -1069.094,E2 -1069.094} C_VEL
LIN {X 0,Y 594.352,Z 259.071,A -85,B 0,C 180,E1 -1071.842,E2 -1071.842} C_VEL
LIN {X 0,Y 594.378,Z 259.071,A -85,B 0,C 180,E1 -1074.572,E2 -1074.572} C_VEL
LIN {X 0,Y 594.371,Z 259.066,A -85,B 0,C 180,E1 -1077.289,E2 -1077.289} C_VEL
LIN {X 0,Y 594.403,Z 259.07,A -85,B 0,C 180,E1 -1080,E2 -1080} C_VEL
LIN {X 0,Y 594.397,Z 259.066,A -85,B 0,C 180,E1 -1082.711,E2 -1082.711} C_VEL
LIN {X 0,Y 594.359,Z 259.069,A -85,B 0,C 180,E1 -1085.428,E2 -1085.428} C_VEL
LIN {X 0,Y 594.377,Z 259.076,A -85,B 0,C 180,E1 -1088.157,E2 -1088.157} C_VEL
LIN {X 0,Y 594.369,Z 259.066,A -85,B 0,C 180,E1 -1091.064,E2 -1091.064} C_VEL
LIN {X 0,Y 594.367,Z 259.072,A -85,B 0,C 180,E1 -1093.679,E2 -1093.679} C_VEL
LIN {X 0,Y 594.373,Z 259.067,A -85,B 0,C 180,E1 -1096.713,E2 -1096.713} C_VEL
LIN {X 0,Y 594.358,Z 259.07,A -85,B 0,C 180,E1 -1099.335,E2 -1099.335} C_VEL
LIN {X 0,Y 594.356,Z 259.072,A -85,B 0,C 180,E1 -1101.504,E2 -1101.504} C_VEL
LIN {X 0,Y 594.388,Z 259.065,A -85,B 0,C 180,E1 -1104.446,E2 -1104.446} C_VEL
LIN {X 0,Y 594.355,Z 259.068,A -85,B 0,C 180,E1 -1106.701,E2 -1106.701} C_VEL
LIN {X 0,Y 594.374,Z 259.067,A -85,B 0,C 180,E1 -1108.999,E2 -1108.999} C_VEL
LIN {X 0,Y 594.374,Z 259.073,A -85,B 0,C 180,E1 -1111.642,E2 -1111.642} C_VEL
LIN {X 0,Y 594.368,Z 259.067,A -85,B 0,C 180,E1 -1114.581,E2 -1114.581} C_VEL
LIN {X 0,Y 594.385,Z 259.073,A -85,B 0,C 180,E1 -1117.608,E2 -1117.608} C_VEL
LIN {X 0,Y 594.363,Z 259.068,A -85,B 0,C 180,E1 -1120.567,E2 -1120.567} C_VEL
LIN {X 0,Y 594.363,Z 259.072,A -85,B 0,C 180,E1 -1123.3,E2 -1123.3} C_VEL
LIN {X 0,Y 594.358,Z 259.07,A -85,B 0,C 180,E1 -1126.161,E2 -1126.161} C_VEL
LIN {X 0,Y 594.373,Z 259.066,A -85,B 0,C 180,E1 -1128.536,E2 -1128.536} C_VEL
LIN {X 0,Y 594.379,Z 259.072,A -85,B 0,C 180,E1 -1131.296,E2 -1131.296} C_VEL
LIN {X 0,Y 594.393,Z 259.07,A -85,B 0,C 180,E1 -1133.759,E2 -1133.759} C_VEL
LIN {X 0,Y 594.374,Z 259.067,A -85,B 0,C 180,E1 -1136.239,E2 -1136.239} C_VEL
LIN {X 0,Y 594.366,Z 259.068,A -85,B 0,C 180,E1 -1138.65,E2 -1138.65} C_VEL
LIN {X 0,Y 594.383,Z 259.07,A -85,B 0,C 180,E1 -1141.042,E2 -1141.042} C_VEL
LIN {X 0,Y 594.379,Z 259.124,A -85,B 0,C 180,E1 -1143.885,E2 -1143.885} C_VEL
LIN {X 0,Y 595.045,Z 262.168,A -85,B 0,C 180,E1 -1144.275,E2 -1144.275} C_VEL
LIN {X 0,Y 594.99,Z 282.913,A -85,B 0,C 180,E1 -1146.691,E2 -1146.691} C_VEL
LIN {X 0,Y 594.82,Z 308.446,A -85,B 0,C 180,E1 -1149.601,E2 -1149.601} C_VEL
LIN {X 0,Y 594.752,Z 322.058,A -85,B 0,C 180,E1 -1151.103,E2 -1151.103} C_VEL
LIN {X 0,Y 595.337,Z 325.943,A -85,B 0,C 180,E1 -1151.17,E2 -1151.17} C_VEL
LIN {X 0,Y 595.084,Z 488.326,A -85,B 0,C 180,E1 -1153.198,E2 -1153.198} C_VEL
LIN {X 0,Y 595.025,Z 503.72,A -85,B 0,C 180,E1 -1153.533,E2 -1153.533} C_VEL
LIN {X 0,Y 594.933,Z 519.053,A -85,B 0,C 180,E1 -1154.015,E2 -1154.015} C_VEL
LIN {X 0,Y 594.857,Z 532.769,A -85,B 0,C 180,E1 -1154.584,E2 -1154.584} C_VEL
LIN {X 0,Y 594.737,Z 546.241,A -85,B 0,C 180,E1 -1155.282,E2 -1155.282} C_VEL
LIN {X 0,Y 594.68,Z 558.797,A -85,B 0,C 180,E1 -1156.075,E2 -1156.075} C_VEL
LIN {X 0,Y 594.56,Z 571.289,A -85,B 0,C 180,E1 -1157.022,E2 -1157.022} C_VEL
LIN {X 0,Y 594.465,Z 582.751,A -85,B 0,C 180,E1 -1158.06,E2 -1158.06} C_VEL
LIN {X 0,Y 594.389,Z 592.392,A -85,B 0,C 180,E1 -1159.095,E2 -1159.095} C_VEL
LIN {X 0,Y 594.366,Z 601.858,A -85,B 0,C 180,E1 -1160.3,E2 -1160.3} C_VEL
LIN {X 0,Y 594.31,Z 609.733,A -85,B 0,C 180,E1 -1161.5,E2 -1161.5} C_VEL
LIN {X 0,Y 594.292,Z 617.09,A -85,B 0,C 180,E1 -1162.867,E2 -1162.867} C_VEL
LIN {X 0,Y 594.296,Z 622.925,A -85,B 0,C 180,E1 -1164.231,E2 -1164.231} C_VEL
LIN {X 0,Y 594.232,Z 626.385,A -85,B 0,C 180,E1 -1165.251,E2 -1165.251} C_VEL
LIN {X 0,Y 594.256,Z 629.888,A -85,B 0,C 180,E1 -1166.61,E2 -1166.61} C_VEL
LIN {X 0,Y 594.24,Z 632.193,A -85,B 0,C 180,E1 -1167.967,E2 -1167.967} C_VEL
LIN {X 0,Y 594.237,Z 633.35,A -85,B 0,C 180,E1 -1169.323,E2 -1169.323} C_VEL
LIN {X 0,Y 594.237,Z 633.35,A -85,B 0,C 180,E1 -1170.678,E2 -1170.678} C_VEL
LIN {X 0,Y 594.24,Z 632.192,A -85,B 0,C 180,E1 -1172.034,E2 -1172.034} C_VEL
LIN {X 0,Y 594.256,Z 629.885,A -85,B 0,C 180,E1 -1173.39,E2 -1173.39} C_VEL
LIN {X 0,Y 594.233,Z 626.383,A -85,B 0,C 180,E1 -1174.749,E2 -1174.749} C_VEL
LIN {X 0,Y 594.275,Z 621.606,A -85,B 0,C 180,E1 -1176.11,E2 -1176.11} C_VEL
LIN {X 0,Y 594.287,Z 615.423,A -85,B 0,C 180,E1 -1177.475,E2 -1177.475} C_VEL
LIN {X 0,Y 594.331,Z 607.649,A -85,B 0,C 180,E1 -1178.843,E2 -1178.843} C_VEL
LIN {X 0,Y 594.387,Z 599.367,A -85,B 0,C 180,E1 -1180.044,E2 -1180.044} C_VEL
LIN {X 0,Y 594.434,Z 589.555,A -85,B 0,C 180,E1 -1181.231,E2 -1181.231} C_VEL
LIN {X 0,Y 594.531,Z 579.187,A -85,B 0,C 180,E1 -1182.286,E2 -1182.286} C_VEL
LIN {X 0,Y 594.582,Z 567.012,A -85,B 0,C 180,E1 -1183.326,E2 -1183.326} C_VEL
LIN {X 0,Y 594.695,Z 555.068,A -85,B 0,C 180,E1 -1184.178,E2 -1184.178} C_VEL
LIN {X 0,Y 594.783,Z 541.516,A -85,B 0,C 180,E1 -1184.98,E2 -1184.98} C_VEL
LIN {X 0,Y 594.906,Z 526.83,A -85,B 0,C 180,E1 -1185.679,E2 -1185.679} C_VEL
LIN {X 0,Y 594.967,Z 512.605,A -85,B 0,C 180,E1 -1186.205,E2 -1186.205} C_VEL
LIN {X 0,Y 595.052,Z 498.092,A -85,B 0,C 180,E1 -1186.603,E2 -1186.603} C_VEL
LIN {X 0,Y 595.07,Z 482.658,A -85,B 0,C 180,E1 -1186.887,E2 -1186.887} C_VEL
LIN {X 0,Y 595.224,Z 324.507,A -85,B 0,C 180,E1 -1188.851,E2 -1188.851} C_VEL
LIN {X 0,Y 594.735,Z 321.653,A -85,B 0,C 180,E1 -1188.914,E2 -1188.914} C_VEL
LIN {X 0,Y 594.887,Z 297.27,A -85,B 0,C 180,E1 -1191.666,E2 -1191.666} C_VEL
LIN {X 0,Y 595.067,Z 271.956,A -85,B 0,C 180,E1 -1194.577,E2 -1194.577} C_VEL
LIN {X 0,Y 595.045,Z 262.162,A -85,B 0,C 180,E1 -1195.725,E2 -1195.725} C_VEL
LIN {X 0,Y 594.372,Z 259.075,A -85,B 0,C 180,E1 -1196.138,E2 -1196.138} C_VEL
LIN {X 0,Y 594.38,Z 259.07,A -85,B 0,C 180,E1 -1198.999,E2 -1198.999} C_VEL
LIN {X 0,Y 594.378,Z 259.066,A -85,B 0,C 180,E1 -1201.643,E2 -1201.643} C_VEL
LIN {X 0,Y 594.374,Z 259.076,A -85,B 0,C 180,E1 -1204.581,E2 -1204.581} C_VEL
LIN {X 0,Y 594.389,Z 259.065,A -85,B 0,C 180,E1 -1207.608,E2 -1207.608} C_VEL
LIN {X 0,Y 594.367,Z 259.076,A -85,B 0,C 180,E1 -1210.568,E2 -1210.568} C_VEL
LIN {X 0,Y 594.354,Z 259.069,A -85,B 0,C 180,E1 -1213.301,E2 -1213.301} C_VEL
LIN {X 0,Y 594.363,Z 259.074,A -85,B 0,C 180,E1 -1216.162,E2 -1216.162} C_VEL
LIN {X 0,Y 594.377,Z 259.073,A -85,B 0,C 180,E1 -1218.536,E2 -1218.536} C_VEL
LIN {X 0,Y 594.372,Z 259.066,A -85,B 0,C 180,E1 -1221.298,E2 -1221.298} C_VEL
LIN {X 0,Y 594.352,Z 259.071,A -85,B 0,C 180,E1 -1223.756,E2 -1223.756} C_VEL
LIN {X 0,Y 594.377,Z 259.076,A -85,B 0,C 180,E1 -1226.239,E2 -1226.239} C_VEL
LIN {X 0,Y 594.367,Z 259.07,A -85,B 0,C 180,E1 -1228.65,E2 -1228.65} C_VEL
LIN {X 0,Y 594.38,Z 259.065,A -85,B 0,C 180,E1 -1231.044,E2 -1231.044} C_VEL
LIN {X 0,Y 594.371,Z 259.075,A -85,B 0,C 180,E1 -1234.056,E2 -1234.056} C_VEL
LIN {X 0,Y 594.374,Z 259.073,A -85,B 0,C 180,E1 -1236.295,E2 -1236.295} C_VEL
LIN {X 0,Y 594.399,Z 259.063,A -85,B 0,C 180,E1 -1239.224,E2 -1239.224} C_VEL
LIN {X 0,Y 594.345,Z 259.08,A -85,B 0,C 180,E1 -1242.095,E2 -1242.095} C_VEL
LIN {X 0,Y 594.355,Z 259.075,A -85,B 0,C 180,E1 -1244.219,E2 -1244.219} C_VEL
LIN {X 0,Y 594.371,Z 259.072,A -85,B 0,C 180,E1 -1246.321,E2 -1246.321} C_VEL
LIN {X 0,Y 594.353,Z 259.068,A -85,B 0,C 180,E1 -1249.094,E2 -1249.094} C_VEL
LIN {X 0,Y 594.381,Z 259.074,A -85,B 0,C 180,E1 -1251.843,E2 -1251.843} C_VEL
LIN {X 0,Y 594.363,Z 259.069,A -85,B 0,C 180,E1 -1254.572,E2 -1254.572} C_VEL
LIN {X 0,Y 594.399,Z 259.065,A -85,B 0,C 180,E1 -1257.289,E2 -1257.289} C_VEL
LIN {X 0,Y 594.409,Z 259.069,A -85,B 0,C 180,E1 -1260,E2 -1260} C_VEL
LIN {X 0,Y 594.375,Z 259.066,A -85,B 0,C 180,E1 -1262.711,E2 -1262.711} C_VEL
LIN {X 0,Y 594.381,Z 259.07,A -85,B 0,C 180,E1 -1265.428,E2 -1265.428} C_VEL
LIN {X 0,Y 594.356,Z 259.072,A -85,B 0,C 180,E1 -1268.158,E2 -1268.158} C_VEL
LIN {X 0,Y 594.37,Z 259.068,A -85,B 0,C 180,E1 -1271.061,E2 -1271.061} C_VEL
LIN {X 0,Y 594.336,Z 259.073,A -85,B 0,C 180,E1 -1274.151,E2 -1274.151} C_VEL
LIN {X 0,Y 594.331,Z 259.074,A -85,B 0,C 180,E1 -1275.278,E2 -1275.278} C_VEL
LIN {X 0,Y 593.658,Z 259.164,A -85,B 0,C 180,E1 -1275.843,E2 -1275.843} C_VEL
LIN {X 0,Y 590.791,Z 259.52,A -85,B 0,C 180,E1 -1276.761,E2 -1276.761} C_VEL
LIN {X 0,Y 588.378,Z 259.822,A -85,B 0,C 180,E1 -1277.499,E2 -1277.499} C_VEL
LIN {X 0,Y 587.354,Z 259.944,A -85,B 0,C 180,E1 -1278.069,E2 -1278.069} C_VEL
LIN {X 0,Y 587.277,Z 259.951,A -85,B 0,C 180,E1 -1278.262,E2 -1278.262} C_VEL
LIN {X 0,Y 587.301,Z 259.95,A -85,B 0,C 180,E1 -1281.039,E2 -1281.039} C_VEL
LIN {X 0,Y 587.283,Z 259.953,A -85,B 0,C 180,E1 -1284.009,E2 -1284.009} C_VEL
LIN {X 0,Y 587.299,Z 259.947,A -85,B 0,C 180,E1 -1286.281,E2 -1286.281} C_VEL
LIN {X 0,Y 587.301,Z 259.95,A -85,B 0,C 180,E1 -1289.124,E2 -1289.124} C_VEL
LIN {X 0,Y 587.297,Z 259.952,A -85,B 0,C 180,E1 -1291.827,E2 -1291.827} C_VEL
LIN {X 0,Y 587.303,Z 259.947,A -85,B 0,C 180,E1 -1294.34,E2 -1294.34} C_VEL
LIN {X 0,Y 587.308,Z 259.953,A -85,B 0,C 180,E1 -1297.611,E2 -1297.611} C_VEL
LIN {X 0,Y 587.276,Z 259.95,A -85,B 0,C 180,E1 -1300.258,E2 -1300.258} C_VEL
LIN {X 0,Y 587.281,Z 259.957,A -85,B 0,C 180,E1 -1303.114,E2 -1303.114} C_VEL
LIN {X 0,Y 587.27,Z 259.951,A -85,B 0,C 180,E1 -1306.044,E2 -1306.044} C_VEL
LIN {X 0,Y 587.268,Z 259.957,A -85,B 0,C 180,E1 -1308.933,E2 -1308.933} C_VEL
LIN {X 0,Y 587.27,Z 259.956,A -85,B 0,C 180,E1 -1311.515,E2 -1311.515} C_VEL
LIN {X 0,Y 587.257,Z 259.953,A -85,B 0,C 180,E1 -1314.097,E2 -1314.097} C_VEL
LIN {X 0,Y 587.293,Z 259.95,A -85,B 0,C 180,E1 -1316.6,E2 -1316.6} C_VEL
LIN {X 0,Y 587.294,Z 259.957,A -85,B 0,C 180,E1 -1319.031,E2 -1319.031} C_VEL
LIN {X 0,Y 587.275,Z 259.956,A -85,B 0,C 180,E1 -1321.4,E2 -1321.4} C_VEL
LIN {X 0,Y 587.295,Z 259.95,A -85,B 0,C 180,E1 -1323.832,E2 -1323.832} C_VEL
LIN {X 0,Y 587.293,Z 259.956,A -85,B 0,C 180,E1 -1326.74,E2 -1326.74} C_VEL
LIN {X 0,Y 587.318,Z 260.041,A -85,B 0,C 180,E1 -1327.693,E2 -1327.693} C_VEL
LIN {X 0,Y 587.809,Z 263.819,A -85,B 0,C 180,E1 -1328.244,E2 -1328.244} C_VEL
LIN {X 0,Y 587.684,Z 283.084,A -85,B 0,C 180,E1 -1330.919,E2 -1330.919} C_VEL
LIN {X 0,Y 588.578,Z 287.905,A -85,B 0,C 180,E1 -1331.016,E2 -1331.016} C_VEL
LIN {X 0,Y 588.292,Z 448.448,A -85,B 0,C 180,E1 -1333.046,E2 -1333.046} C_VEL
LIN {X 0,Y 588.199,Z 464.465,A -85,B 0,C 180,E1 -1333.403,E2 -1333.403} C_VEL
LIN {X 0,Y 588.083,Z 479.026,A -85,B 0,C 180,E1 -1333.867,E2 -1333.867} C_VEL
LIN {X 0,Y 587.996,Z 493.697,A -85,B 0,C 180,E1 -1334.488,E2 -1334.488} C_VEL
LIN {X 0,Y 587.846,Z 507.002,A -85,B 0,C 180,E1 -1335.193,E2 -1335.193} C_VEL
LIN {X 0,Y 587.736,Z 520.169,A -85,B 0,C 180,E1 -1336.047,E2 -1336.047} C_VEL
LIN {X 0,Y 587.559,Z 532.861,A -85,B 0,C 180,E1 -1337.039,E2 -1337.039} C_VEL
LIN {X 0,Y 587.473,Z 544.064,A -85,B 0,C 180,E1 -1338.09,E2 -1338.09} C_VEL
LIN {X 0,Y 587.383,Z 554.948,A -85,B 0,C 180,E1 -1339.312,E2 -1339.312} C_VEL
LIN {X 0,Y 587.285,Z 563.992,A -85,B 0,C 180,E1 -1340.529,E2 -1340.529} C_VEL
LIN {X 0,Y 587.259,Z 571.486,A -85,B 0,C 180,E1 -1341.743,E2 -1341.743} C_VEL
LIN {X 0,Y 587.208,Z 578.491,A -85,B 0,C 180,E1 -1343.126,E2 -1343.126} C_VEL
LIN {X 0,Y 587.198,Z 584,A -85,B 0,C 180,E1 -1344.505,E2 -1344.505} C_VEL
LIN {X 0,Y 587.17,Z 588.172,A -85,B 0,C 180,E1 -1345.881,E2 -1345.881} C_VEL
LIN {X 0,Y 587.127,Z 591.113,A -85,B 0,C 180,E1 -1347.255,E2 -1347.255} C_VEL
LIN {X 0,Y 587.143,Z 592.88,A -85,B 0,C 180,E1 -1348.628,E2 -1348.628} C_VEL
LIN {X 0,Y 587.135,Z 593.496,A -85,B 0,C 180,E1 -1350,E2 -1350} C_VEL
LIN {X 0,Y 587.146,Z 592.944,A -85,B 0,C 180,E1 -1351.371,E2 -1351.371} C_VEL
LIN {X 0,Y 587.129,Z 591.26,A -85,B 0,C 180,E1 -1352.744,E2 -1352.744} C_VEL
LIN {X 0,Y 587.169,Z 588.406,A -85,B 0,C 180,E1 -1354.118,E2 -1354.118} C_VEL
LIN {X 0,Y 587.198,Z 584.324,A -85,B 0,C 180,E1 -1355.494,E2 -1355.494} C_VEL
LIN {X 0,Y 587.207,Z 578.914,A -85,B 0,C 180,E1 -1356.874,E2 -1356.874} C_VEL
LIN {X 0,Y 587.254,Z 572.015,A -85,B 0,C 180,E1 -1358.257,E2 -1358.257} C_VEL
LIN {X 0,Y 587.286,Z 563.411,A -85,B 0,C 180,E1 -1359.644,E2 -1359.644} C_VEL
LIN {X 0,Y 587.367,Z 554.261,A -85,B 0,C 180,E1 -1360.862,E2 -1360.862} C_VEL
LIN {X 0,Y 587.447,Z 544.933,A -85,B 0,C 180,E1 -1361.91,E2 -1361.91} C_VEL
LIN {X 0,Y 587.589,Z 532.892,A -85,B 0,C 180,E1 -1363.047,E2 -1363.047} C_VEL
LIN {X 0,Y 587.71,Z 519.799,A -85,B 0,C 180,E1 -1364.069,E2 -1364.069} C_VEL
LIN {X 0,Y 587.809,Z 507.04,A -85,B 0,C 180,E1 -1364.895,E2 -1364.895} C_VEL
LIN {X 0,Y 587.987,Z 493.738,A -85,B 0,C 180,E1 -1365.601,E2 -1365.601} C_VEL
LIN {X 0,Y 588.069,Z 479.063,A -85,B 0,C 180,E1 -1366.221,E2 -1366.221} C_VEL
LIN {X 0,Y 588.224,Z 463.344,A -85,B 0,C 180,E1 -1366.718,E2 -1366.718} C_VEL
LIN {X 0,Y 588.282,Z 448.505,A -85,B 0,C 180,E1 -1367.044,E2 -1367.044} C_VEL
LIN {X 0,Y 588.589,Z 287.636,A -85,B 0,C 180,E1 -1369.077,E2 -1369.077} C_VEL
LIN {X 0,Y 587.702,Z 283.097,A -85,B 0,C 180,E1 -1369.169,E2 -1369.169} C_VEL
LIN {X 0,Y 587.808,Z 263.15,A -85,B 0,C 180,E1 -1371.94,E2 -1371.94} C_VEL
LIN {X 0,Y 587.329,Z 259.951,A -85,B 0,C 180,E1 -1372.421,E2 -1372.421} C_VEL
LIN {X 0,Y 587.305,Z 259.951,A -85,B 0,C 180,E1 -1375.518,E2 -1375.518} C_VEL
LIN {X 0,Y 587.289,Z 259.95,A -85,B 0,C 180,E1 -1377.82,E2 -1377.82} C_VEL
LIN {X 0,Y 587.304,Z 259.951,A -85,B 0,C 180,E1 -1380.504,E2 -1380.504} C_VEL
LIN {X 0,Y 587.278,Z 259.959,A -85,B 0,C 180,E1 -1383.102,E2 -1383.102} C_VEL
LIN {X 0,Y 587.266,Z 259.953,A -85,B 0,C 180,E1 -1385.533,E2 -1385.533} C_VEL
LIN {X 0,Y 587.304,Z 259.948,A -85,B 0,C 180,E1 -1387.834,E2 -1387.834} C_VEL
LIN {X 0,Y 587.294,Z 259.95,A -85,B 0,C 180,E1 -1390.256,E2 -1390.256} C_VEL
LIN {X 0,Y 587.281,Z 259.954,A -85,B 0,C 180,E1 -1393.115,E2 -1393.115} C_VEL
LIN {X 0,Y 587.284,Z 259.95,A -85,B 0,C 180,E1 -1396.046,E2 -1396.046} C_VEL
LIN {X 0,Y 587.287,Z 259.956,A -85,B 0,C 180,E1 -1398.93,E2 -1398.93} C_VEL
LIN {X 0,Y 587.264,Z 259.952,A -85,B 0,C 180,E1 -1401.515,E2 -1401.515} C_VEL
LIN {X 0,Y 587.249,Z 259.953,A -85,B 0,C 180,E1 -1404.097,E2 -1404.097} C_VEL
LIN {X 0,Y 587.3,Z 259.957,A -85,B 0,C 180,E1 -1406.601,E2 -1406.601} C_VEL
LIN {X 0,Y 587.291,Z 259.952,A -85,B 0,C 180,E1 -1409.031,E2 -1409.031} C_VEL
LIN {X 0,Y 587.265,Z 259.952,A -85,B 0,C 180,E1 -1411.4,E2 -1411.4} C_VEL
LIN {X 0,Y 587.292,Z 259.949,A -85,B 0,C 180,E1 -1413.832,E2 -1413.832} C_VEL
LIN {X 0,Y 587.283,Z 259.956,A -85,B 0,C 180,E1 -1416.74,E2 -1416.74} C_VEL
LIN {X 0,Y 587.296,Z 259.949,A -85,B 0,C 180,E1 -1419.694,E2 -1419.694} C_VEL
LIN {X 0,Y 587.272,Z 259.952,A -85,B 0,C 180,E1 -1421.872,E2 -1421.872} C_VEL
LIN {X 0,Y 587.299,Z 259.952,A -85,B 0,C 180,E1 -1424.736,E2 -1424.736} C_VEL
LIN {X 0,Y 587.273,Z 259.954,A -85,B 0,C 180,E1 -1426.857,E2 -1426.857} C_VEL
LIN {X 0,Y 587.337,Z 259.944,A -85,B 0,C 180,E1 -1428.962,E2 -1428.962} C_VEL
LIN {X 0,Y 587.316,Z 259.947,A -85,B 0,C 180,E1 -1431.744,E2 -1431.744} C_VEL
LIN {X 0,Y 587.343,Z 259.948,A -85,B 0,C 180,E1 -1434.507,E2 -1434.507} C_VEL
LIN {X 0,Y 587.341,Z 259.942,A -85,B 0,C 180,E1 -1437.257,E2 -1437.257} C_VEL
LIN {X 0,Y 587.372,Z 259.945,A -85,B 0,C 180,E1 -1440,E2 -1440} C_VEL
LIN {X 0,Y 587.36,Z 259.942,A -85,B 0,C 180,E1 -1442.743,E2 -1442.743} C_VEL
LIN {X 0,Y 587.328,Z 259.945,A -85,B 0,C 180,E1 -1445.493,E2 -1445.493} C_VEL
LIN {X 0,Y 587.337,Z 259.951,A -85,B 0,C 180,E1 -1448.256,E2 -1448.256} C_VEL
LIN {X 0,Y 587.348,Z 259.941,A -85,B 0,C 180,E1 -1451.134,E2 -1451.134} C_VEL
LIN {X 0,Y 587.364,Z 259.945,A -85,B 0,C 180,E1 -1454.26,E2 -1454.26} C_VEL
LIN {X 0,Y 587.307,Z 259.949,A -85,B 0,C 180,E1 -1457.407,E2 -1457.407} C_VEL
LIN {X 0,Y 587.306,Z 259.951,A -85,B 0,C 180,E1 -1459.576,E2 -1459.576} C_VEL
LIN {X 0,Y 587.314,Z 259.954,A -85,B 0,C 180,E1 -1461.775,E2 -1461.775} C_VEL
LIN {X 0,Y 587.345,Z 259.94,A -85,B 0,C 180,E1 -1464.759,E2 -1464.759} C_VEL
LIN {X 0,Y 587.3,Z 259.947,A -85,B 0,C 180,E1 -1467.048,E2 -1467.048} C_VEL
LIN {X 0,Y 587.342,Z 259.946,A -85,B 0,C 180,E1 -1469.38,E2 -1469.38} C_VEL
LIN {X 0,Y 587.342,Z 259.95,A -85,B 0,C 180,E1 -1471.835,E2 -1471.835} C_VEL
LIN {X 0,Y 587.341,Z 259.944,A -85,B 0,C 180,E1 -1474.347,E2 -1474.347} C_VEL
LIN {X 0,Y 587.347,Z 259.941,A -85,B 0,C 180,E1 -1476.747,E2 -1476.747} C_VEL
LIN {X 0,Y 587.327,Z 259.949,A -85,B 0,C 180,E1 -1479.361,E2 -1479.361} C_VEL
LIN {X 0,Y 587.334,Z 259.947,A -85,B 0,C 180,E1 -1482.108,E2 -1482.108} C_VEL
LIN {X 0,Y 587.287,Z 259.952,A -85,B 0,C 180,E1 -1485.086,E2 -1485.086} C_VEL
LIN {X 0,Y 587.338,Z 259.947,A -85,B 0,C 180,E1 -1487.926,E2 -1487.926} C_VEL
LIN {X 0,Y 587.32,Z 259.948,A -85,B 0,C 180,E1 -1491.06,E2 -1491.06} C_VEL
LIN {X 0,Y 587.351,Z 259.948,A -85,B 0,C 180,E1 -1493.292,E2 -1493.292} C_VEL
LIN {X 0,Y 587.36,Z 259.946,A -85,B 0,C 180,E1 -1495.78,E2 -1495.78} C_VEL
LIN {X 0,Y 587.341,Z 259.944,A -85,B 0,C 180,E1 -1498.231,E2 -1498.231} C_VEL
LIN {X 0,Y 587.35,Z 259.945,A -85,B 0,C 180,E1 -1500.867,E2 -1500.867} C_VEL
LIN {X 0,Y 587.347,Z 259.974,A -85,B 0,C 180,E1 -1503.65,E2 -1503.65} C_VEL
LIN {X 0,Y 588.317,Z 265.36,A -85,B 0,C 180,E1 -1504.34,E2 -1504.34} C_VEL
LIN {X 0,Y 588.101,Z 290.157,A -85,B 0,C 180,E1 -1507.246,E2 -1507.246} C_VEL
LIN {X 0,Y 587.868,Z 316.425,A -85,B 0,C 180,E1 -1510.262,E2 -1510.262} C_VEL
LIN {X 0,Y 587.805,Z 321.744,A -85,B 0,C 180,E1 -1510.865,E2 -1510.865} C_VEL
LIN {X 0,Y 588.617,Z 326.023,A -85,B 0,C 180,E1 -1510.948,E2 -1510.948} C_VEL
LIN {X 0,Y 588.294,Z 488.482,A -85,B 0,C 180,E1 -1513.001,E2 -1513.001} C_VEL
LIN {X 0,Y 588.216,Z 504.493,A -85,B 0,C 180,E1 -1513.359,E2 -1513.359} C_VEL
LIN {X 0,Y 588.071,Z 519.052,A -85,B 0,C 180,E1 -1513.823,E2 -1513.823} C_VEL
LIN {X 0,Y 587.988,Z 532.772,A -85,B 0,C 180,E1 -1514.399,E2 -1514.399} C_VEL
LIN {X 0,Y 587.836,Z 546.244,A -85,B 0,C 180,E1 -1515.105,E2 -1515.105} C_VEL
LIN {X 0,Y 587.74,Z 559.118,A -85,B 0,C 180,E1 -1515.93,E2 -1515.93} C_VEL
LIN {X 0,Y 587.583,Z 571.291,A -85,B 0,C 180,E1 -1516.865,E2 -1516.865} C_VEL
LIN {X 0,Y 587.453,Z 582.751,A -85,B 0,C 180,E1 -1517.915,E2 -1517.915} C_VEL
LIN {X 0,Y 587.349,Z 592.393,A -85,B 0,C 180,E1 -1518.963,E2 -1518.963} C_VEL
LIN {X 0,Y 587.304,Z 601.858,A -85,B 0,C 180,E1 -1520.182,E2 -1520.182} C_VEL
LIN {X 0,Y 587.264,Z 609.734,A -85,B 0,C 180,E1 -1521.397,E2 -1521.397} C_VEL
LIN {X 0,Y 587.215,Z 617.09,A -85,B 0,C 180,E1 -1522.781,E2 -1522.781} C_VEL
LIN {X 0,Y 587.224,Z 622.925,A -85,B 0,C 180,E1 -1524.162,E2 -1524.162} C_VEL
LIN {X 0,Y 587.136,Z 626.385,A -85,B 0,C 180,E1 -1525.194,E2 -1525.194} C_VEL
LIN {X 0,Y 587.179,Z 629.888,A -85,B 0,C 180,E1 -1526.569,E2 -1526.569} C_VEL
LIN {X 0,Y 587.138,Z 632.194,A -85,B 0,C 180,E1 -1527.942,E2 -1527.942} C_VEL
LIN {X 0,Y 587.137,Z 633.35,A -85,B 0,C 180,E1 -1529.314,E2 -1529.314} C_VEL
LIN {X 0,Y 587.137,Z 633.349,A -85,B 0,C 180,E1 -1530.686,E2 -1530.686} C_VEL
LIN {X 0,Y 587.138,Z 632.192,A -85,B 0,C 180,E1 -1532.058,E2 -1532.058} C_VEL
LIN {X 0,Y 587.179,Z 629.886,A -85,B 0,C 180,E1 -1533.431,E2 -1533.431} C_VEL
LIN {X 0,Y 587.136,Z 626.383,A -85,B 0,C 180,E1 -1534.807,E2 -1534.807} C_VEL
LIN {X 0,Y 587.178,Z 621.607,A -85,B 0,C 180,E1 -1536.184,E2 -1536.184} C_VEL
LIN {X 0,Y 587.23,Z 615.422,A -85,B 0,C 180,E1 -1537.565,E2 -1537.565} C_VEL
LIN {X 0,Y 587.267,Z 607.648,A -85,B 0,C 180,E1 -1538.951,E2 -1538.951} C_VEL
LIN {X 0,Y 587.351,Z 599.367,A -85,B 0,C 180,E1 -1540.166,E2 -1540.166} C_VEL
LIN {X 0,Y 587.4,Z 589.391,A -85,B 0,C 180,E1 -1541.386,E2 -1541.386} C_VEL
LIN {X 0,Y 587.522,Z 579.186,A -85,B 0,C 180,E1 -1542.435,E2 -1542.435} C_VEL
LIN {X 0,Y 587.629,Z 567.013,A -85,B 0,C 180,E1 -1543.487,E2 -1543.487} C_VEL
LIN {X 0,Y 587.775,Z 554.05,A -85,B 0,C 180,E1 -1544.416,E2 -1544.416} C_VEL
LIN {X 0,Y 587.889,Z 539.858,A -85,B 0,C 180,E1 -1545.249,E2 -1545.249} C_VEL
LIN {X 0,Y 588.051,Z 525.786,A -85,B 0,C 180,E1 -1545.911,E2 -1545.911} C_VEL
LIN {X 0,Y 588.171,Z 511.29,A -85,B 0,C 180,E1 -1546.442,E2 -1546.442} C_VEL
LIN {X 0,Y 588.281,Z 496.249,A -85,B 0,C 180,E1 -1546.845,E2 -1546.845} C_VEL
LIN {X 0,Y 588.323,Z 481.032,A -85,B 0,C 180,E1 -1547.111,E2 -1547.111} C_VEL
LIN {X 0,Y 588.531,Z 325.414,A -85,B 0,C 180,E1 -1549.062,E2 -1549.062} C_VEL
LIN {X 0,Y 587.823,Z 321.685,A -85,B 0,C 180,E1 -1549.141,E2 -1549.141} C_VEL
LIN {X 0,Y 588.027,Z 297.27,A -85,B 0,C 180,E1 -1551.932,E2 -1551.932} C_VEL
LIN {X 0,Y 588.263,Z 272.866,A -85,B 0,C 180,E1 -1554.773,E2 -1554.773} C_VEL
LIN {X 0,Y 588.213,Z 263.758,A -85,B 0,C 180,E1 -1555.856,E2 -1555.856} C_VEL
LIN {X 0,Y 587.347,Z 259.951,A -85,B 0,C 180,E1 -1556.374,E2 -1556.374} C_VEL
LIN {X 0,Y 587.346,Z 259.943,A -85,B 0,C 180,E1 -1559.38,E2 -1559.38} C_VEL
LIN {X 0,Y 587.345,Z 259.943,A -85,B 0,C 180,E1 -1561.836,E2 -1561.836} C_VEL
LIN {X 0,Y 587.342,Z 259.95,A -85,B 0,C 180,E1 -1564.347,E2 -1564.347} C_VEL
LIN {X 0,Y 587.344,Z 259.942,A -85,B 0,C 180,E1 -1567.608,E2 -1567.608} C_VEL
LIN {X 0,Y 587.312,Z 259.952,A -85,B 0,C 180,E1 -1570.255,E2 -1570.255} C_VEL
LIN {X 0,Y 587.306,Z 259.948,A -85,B 0,C 180,E1 -1573.117,E2 -1573.117} C_VEL
LIN {X 0,Y 587.315,Z 259.95,A -85,B 0,C 180,E1 -1576.049,E2 -1576.049} C_VEL
LIN {X 0,Y 587.334,Z 259.945,A -85,B 0,C 180,E1 -1578.926,E2 -1578.926} C_VEL
LIN {X 0,Y 587.322,Z 259.945,A -85,B 0,C 180,E1 -1581.52,E2 -1581.52} C_VEL
LIN {X 0,Y 587.286,Z 259.956,A -85,B 0,C 180,E1 -1584.1,E2 -1584.1} C_VEL
LIN {X 0,Y 587.335,Z 259.947,A -85,B 0,C 180,E1 -1586.603,E2 -1586.603} C_VEL
LIN {X 0,Y 587.337,Z 259.943,A -85,B 0,C 180,E1 -1589.491,E2 -1589.491} C_VEL
LIN {X 0,Y 587.307,Z 259.957,A -85,B 0,C 180,E1 -1592.18,E2 -1592.18} C_VEL
LIN {X 0,Y 587.35,Z 259.941,A -85,B 0,C 180,E1 -1595.241,E2 -1595.241} C_VEL
LIN {X 0,Y 587.319,Z 259.954,A -85,B 0,C 180,E1 -1598.226,E2 -1598.226} C_VEL
LIN {X 0,Y 587.339,Z 259.942,A -85,B 0,C 180,E1 -1601.151,E2 -1601.151} C_VEL
LIN {X 0,Y 587.312,Z 259.956,A -85,B 0,C 180,E1 -1604.025,E2 -1604.025} C_VEL
LIN {X 0,Y 587.355,Z 259.949,A -85,B 0,C 180,E1 -1606.154,E2 -1606.154} C_VEL
LIN {X 0,Y 587.343,Z 259.941,A -85,B 0,C 180,E1 -1608.963,E2 -1608.963} C_VEL
LIN {X 0,Y 587.341,Z 259.949,A -85,B 0,C 180,E1 -1611.744,E2 -1611.744} C_VEL
LIN {X 0,Y 587.332,Z 259.945,A -85,B 0,C 180,E1 -1614.507,E2 -1614.507} C_VEL
LIN {X 0,Y 587.363,Z 259.941,A -85,B 0,C 180,E1 -1617.257,E2 -1617.257} C_VEL
LIN {X 0,Y 587.378,Z 259.945,A -85,B 0,C 180,E1 -1620,E2 -1620} C_VEL
LIN {X 0,Y 587.345,Z 259.942,A -85,B 0,C 180,E1 -1622.743,E2 -1622.743} C_VEL
LIN {X 0,Y 587.346,Z 259.947,A -85,B 0,C 180,E1 -1625.493,E2 -1625.493} C_VEL
LIN {X 0,Y 587.318,Z 259.948,A -85,B 0,C 180,E1 -1628.256,E2 -1628.256} C_VEL
LIN {X 0,Y 587.336,Z 259.944,A -85,B 0,C 180,E1 -1631.124,E2 -1631.124} C_VEL
LIN {X 0,Y 587.306,Z 259.948,A -85,B 0,C 180,E1 -1634.235,E2 -1634.235} C_VEL
LIN {X 0,Y 587.297,Z 259.948,A -85,B 0,C 180,E1 -1636.795,E2 -1636.795} C_VEL
LIN {X 0,Y 587.277,Z 259.951,A -85,B 0,C 180,E1 -1638.262,E2 -1638.262} C_VEL
LIN {X 0,Y 586.625,Z 260.033,A -85,B 0,C 180,E1 -1638.834,E2 -1638.834} C_VEL
LIN {X 0,Y 583.772,Z 260.395,A -85,B 0,C 180,E1 -1639.762,E2 -1639.762} C_VEL
LIN {X 0,Y 581.363,Z 260.691,A -85,B 0,C 180,E1 -1640.51,E2 -1640.51} C_VEL
LIN {X 0,Y 580.343,Z 260.817,A -85,B 0,C 180,E1 -1641.086,E2 -1641.086} C_VEL
LIN {X 0,Y 580.269,Z 260.829,A -85,B 0,C 180,E1 -1641.281,E2 -1641.281} C_VEL
LIN {X 0,Y 580.247,Z 260.827,A -85,B 0,C 180,E1 -1644.319,E2 -1644.319} C_VEL
LIN {X 0,Y 580.242,Z 260.826,A -85,B 0,C 180,E1 -1646.625,E2 -1646.625} C_VEL
LIN {X 0,Y 580.25,Z 260.83,A -85,B 0,C 180,E1 -1649.3,E2 -1649.3} C_VEL
LIN {X 0,Y 580.271,Z 260.824,A -85,B 0,C 180,E1 -1652.202,E2 -1652.202} C_VEL
LIN {X 0,Y 580.261,Z 260.825,A -85,B 0,C 180,E1 -1654.698,E2 -1654.698} C_VEL
LIN {X 0,Y 580.267,Z 260.832,A -85,B 0,C 180,E1 -1657.271,E2 -1657.271} C_VEL
LIN {X 0,Y 580.239,Z 260.827,A -85,B 0,C 180,E1 -1660.264,E2 -1660.264} C_VEL
LIN {X 0,Y 580.243,Z 260.828,A -85,B 0,C 180,E1 -1662.71,E2 -1662.71} C_VEL
LIN {X 0,Y 580.228,Z 260.833,A -85,B 0,C 180,E1 -1665.613,E2 -1665.613} C_VEL
LIN {X 0,Y 580.207,Z 260.831,A -85,B 0,C 180,E1 -1668.224,E2 -1668.224} C_VEL
LIN {X 0,Y 580.236,Z 260.833,A -85,B 0,C 180,E1 -1670.961,E2 -1670.961} C_VEL
LIN {X 0,Y 580.229,Z 260.832,A -85,B 0,C 180,E1 -1673.593,E2 -1673.593} C_VEL
LIN {X 0,Y 580.254,Z 260.825,A -85,B 0,C 180,E1 -1676.141,E2 -1676.141} C_VEL
LIN {X 0,Y 580.238,Z 260.83,A -85,B 0,C 180,E1 -1678.612,E2 -1678.612} C_VEL
LIN {X 0,Y 580.247,Z 260.835,A -85,B 0,C 180,E1 -1681.021,E2 -1681.021} C_VEL
LIN {X 0,Y 580.25,Z 260.829,A -85,B 0,C 180,E1 -1683.675,E2 -1683.675} C_VEL
LIN {X 0,Y 580.243,Z 260.831,A -85,B 0,C 180,E1 -1686.44,E2 -1686.44} C_VEL
LIN {X 0,Y 580.277,Z 260.866,A -85,B 0,C 180,E1 -1687.525,E2 -1687.525} C_VEL
LIN {X 0,Y 580.902,Z 265.139,A -85,B 0,C 180,E1 -1688.159,E2 -1688.159} C_VEL
LIN {X 0,Y 580.741,Z 283.112,A -85,B 0,C 180,E1 -1690.685,E2 -1690.685} C_VEL
LIN {X 0,Y 581.887,Z 288.865,A -85,B 0,C 180,E1 -1690.801,E2 -1690.801} C_VEL
LIN {X 0,Y 581.517,Z 448.298,A -85,B 0,C 180,E1 -1692.839,E2 -1692.839} C_VEL
LIN {X 0,Y 581.411,Z 463.71,A -85,B 0,C 180,E1 -1693.18,E2 -1693.18} C_VEL
LIN {X 0,Y 581.234,Z 479.04,A -85,B 0,C 180,E1 -1693.672,E2 -1693.672} C_VEL
LIN {X 0,Y 581.118,Z 493.707,A -85,B 0,C 180,E1 -1694.3,E2 -1694.3} C_VEL
LIN {X 0,Y 580.926,Z 507.014,A -85,B 0,C 180,E1 -1695.013,E2 -1695.013} C_VEL
LIN {X 0,Y 580.793,Z 520.365,A -85,B 0,C 180,E1 -1695.89,E2 -1695.89} C_VEL
LIN {X 0,Y 580.593,Z 532.869,A -85,B 0,C 180,E1 -1696.881,E2 -1696.881} C_VEL
LIN {X 0,Y 580.461,Z 544.07,A -85,B 0,C 180,E1 -1697.944,E2 -1697.944} C_VEL
LIN {X 0,Y 580.337,Z 555.11,A -85,B 0,C 180,E1 -1699.201,E2 -1699.201} C_VEL
LIN {X 0,Y 580.239,Z 563.995,A -85,B 0,C 180,E1 -1700.413,E2 -1700.413} C_VEL
LIN {X 0,Y 580.196,Z 571.488,A -85,B 0,C 180,E1 -1701.642,E2 -1701.642} C_VEL
LIN {X 0,Y 580.139,Z 578.493,A -85,B 0,C 180,E1 -1703.042,E2 -1703.042} C_VEL
LIN {X 0,Y 580.127,Z 584.002,A -85,B 0,C 180,E1 -1704.438,E2 -1704.438} C_VEL
LIN {X 0,Y 580.088,Z 588.173,A -85,B 0,C 180,E1 -1705.831,E2 -1705.831} C_VEL
LIN {X 0,Y 580.038,Z 591.113,A -85,B 0,C 180,E1 -1707.222,E2 -1707.222} C_VEL
LIN {X 0,Y 580.043,Z 592.88,A -85,B 0,C 180,E1 -1708.611,E2 -1708.611} C_VEL
LIN {X 0,Y 580.035,Z 593.496,A -85,B 0,C 180,E1 -1710,E2 -1710} C_VEL
LIN {X 0,Y 580.045,Z 592.943,A -85,B 0,C 180,E1 -1711.388,E2 -1711.388} C_VEL
LIN {X 0,Y 580.04,Z 591.26,A -85,B 0,C 180,E1 -1712.778,E2 -1712.778} C_VEL
LIN {X 0,Y 580.088,Z 588.406,A -85,B 0,C 180,E1 -1714.168,E2 -1714.168} C_VEL
LIN {X 0,Y 580.123,Z 584.322,A -85,B 0,C 180,E1 -1715.561,E2 -1715.561} C_VEL
LIN {X 0,Y 580.138,Z 578.911,A -85,B 0,C 180,E1 -1716.958,E2 -1716.958} C_VEL
LIN {X 0,Y 580.189,Z 572.011,A -85,B 0,C 180,E1 -1718.358,E2 -1718.358} C_VEL
LIN {X 0,Y 580.235,Z 563.406,A -85,B 0,C 180,E1 -1719.763,E2 -1719.763} C_VEL
LIN {X 0,Y 580.308,Z 553.831,A -85,B 0,C 180,E1 -1721.047,E2 -1721.047} C_VEL
LIN {X 0,Y 580.472,Z 543.202,A -85,B 0,C 180,E1 -1722.232,E2 -1722.232} C_VEL
LIN {X 0,Y 580.606,Z 531.828,A -85,B 0,C 180,E1 -1723.296,E2 -1723.296} C_VEL
LIN {X 0,Y 580.759,Z 519.075,A -85,B 0,C 180,E1 -1724.291,E2 -1724.291} C_VEL
LIN {X 0,Y 580.924,Z 505.466,A -85,B 0,C 180,E1 -1725.166,E2 -1725.166} C_VEL
LIN {X 0,Y 581.115,Z 491.79,A -85,B 0,C 180,E1 -1725.88,E2 -1725.88} C_VEL
LIN {X 0,Y 581.257,Z 477.799,A -85,B 0,C 180,E1 -1726.462,E2 -1726.462} C_VEL
LIN {X 0,Y 581.458,Z 462.791,A -85,B 0,C 180,E1 -1726.932,E2 -1726.932} C_VEL
LIN {X 0,Y 581.499,Z 448.475,A -85,B 0,C 180,E1 -1727.249,E2 -1727.249} C_VEL
LIN {X 0,Y 581.793,Z 288.159,A -85,B 0,C 180,E1 -1729.302,E2 -1729.302} C_VEL
LIN {X 0,Y 580.744,Z 283.078,A -85,B 0,C 180,E1 -1729.41,E2 -1729.41} C_VEL
LIN {X 0,Y 580.885,Z 264.461,A -85,B 0,C 180,E1 -1732.028,E2 -1732.028} C_VEL
LIN {X 0,Y 580.299,Z 260.828,A -85,B 0,C 180,E1 -1732.59,E2 -1732.59} C_VEL
LIN {X 0,Y 580.271,Z 260.834,A -85,B 0,C 180,E1 -1735.081,E2 -1735.081} C_VEL
LIN {X 0,Y 580.242,Z 260.828,A -85,B 0,C 180,E1 -1737.848,E2 -1737.848} C_VEL
LIN {X 0,Y 580.254,Z 260.832,A -85,B 0,C 180,E1 -1740.689,E2 -1740.689} C_VEL
LIN {X 0,Y 580.241,Z 260.832,A -85,B 0,C 180,E1 -1743.307,E2 -1743.307} C_VEL
LIN {X 0,Y 580.218,Z 260.83,A -85,B 0,C 180,E1 -1745.752,E2 -1745.752} C_VEL
LIN {X 0,Y 580.271,Z 260.825,A -85,B 0,C 180,E1 -1748.147,E2 -1748.147} C_VEL
LIN {X 0,Y 580.268,Z 260.834,A -85,B 0,C 180,E1 -1750.846,E2 -1750.846} C_VEL
LIN {X 0,Y 580.223,Z 260.829,A -85,B 0,C 180,E1 -1753.663,E2 -1753.663} C_VEL
LIN {X 0,Y 580.222,Z 260.837,A -85,B 0,C 180,E1 -1756.615,E2 -1756.615} C_VEL
LIN {X 0,Y 580.236,Z 260.831,A -85,B 0,C 180,E1 -1759.151,E2 -1759.151} C_VEL
LIN {X 0,Y 580.233,Z 260.828,A -85,B 0,C 180,E1 -1761.934,E2 -1761.934} C_VEL
LIN {X 0,Y 580.203,Z 260.835,A -85,B 0,C 180,E1 -1764.449,E2 -1764.449} C_VEL
LIN {X 0,Y 580.238,Z 260.832,A -85,B 0,C 180,E1 -1766.972,E2 -1766.972} C_VEL
LIN {X 0,Y 580.248,Z 260.826,A -85,B 0,C 180,E1 -1769.422,E2 -1769.422} C_VEL
LIN {X 0,Y 580.236,Z 260.831,A -85,B 0,C 180,E1 -1772.153,E2 -1772.153} C_VEL
LIN {X 0,Y 580.244,Z 260.83,A -85,B 0,C 180,E1 -1774.917,E2 -1774.917} C_VEL
LIN {X 0,Y 580.245,Z 260.827,A -85,B 0,C 180,E1 -1777.195,E2 -1777.195} C_VEL
LIN {X 0,Y 580.24,Z 260.827,A -85,B 0,C 180,E1 -1779.436,E2 -1779.436} C_VEL
LIN {X 0,Y 580.232,Z 260.827,A -85,B 0,C 180,E1 -1781.644,E2 -1781.644} C_VEL
LIN {X 0,Y 580.265,Z 260.831,A -85,B 0,C 180,E1 -1784.546,E2 -1784.546} C_VEL
LIN {X 0,Y 580.264,Z 260.824,A -85,B 0,C 180,E1 -1787.408,E2 -1787.408} C_VEL
LIN {X 0,Y 580.264,Z 260.824,A -85,B 0,C 180,E1 -1789.533,E2 -1789.533} C_VEL
LIN {X 0,Y 580.286,Z 260.831,A -85,B 0,C 180,E1 -1792.344,E2 -1792.344} C_VEL
LIN {X 0,Y 580.303,Z 260.819,A -85,B 0,C 180,E1 -1795.137,E2 -1795.137} C_VEL
LIN {X 0,Y 580.324,Z 260.821,A -85,B 0,C 180,E1 -1797.918,E2 -1797.918} C_VEL
LIN {X 0,Y 580.354,Z 260.814,A -85,B 0,C 180,E1 -1800.694,E2 -1800.694} C_VEL
LIN {X 0,Y 580.325,Z 260.818,A -85,B 0,C 180,E1 -1802.777,E2 -1802.777} C_VEL
LIN {X 0,Y 580.297,Z 260.821,A -85,B 0,C 180,E1 -1805.56,E2 -1805.56} C_VEL
LIN {X 0,Y 580.305,Z 260.825,A -85,B 0,C 180,E1 -1808.356,E2 -1808.356} C_VEL
LIN {X 0,Y 580.3,Z 260.819,A -85,B 0,C 180,E1 -1811.191,E2 -1811.191} C_VEL
LIN {X 0,Y 580.32,Z 260.827,A -85,B 0,C 180,E1 -1814.017,E2 -1814.017} C_VEL
LIN {X 0,Y 580.312,Z 260.818,A -85,B 0,C 180,E1 -1816.914,E2 -1816.914} C_VEL
LIN {X 0,Y 580.281,Z 260.83,A -85,B 0,C 180,E1 -1819.823,E2 -1819.823} C_VEL
LIN {X 0,Y 580.266,Z 260.831,A -85,B 0,C 180,E1 -1822.053,E2 -1822.053} C_VEL
LIN {X 0,Y 580.3,Z 260.817,A -85,B 0,C 180,E1 -1825.08,E2 -1825.08} C_VEL
LIN {X 0,Y 580.278,Z 260.827,A -85,B 0,C 180,E1 -1828.187,E2 -1828.187} C_VEL
LIN {X 0,Y 580.28,Z 260.821,A -85,B 0,C 180,E1 -1830.694,E2 -1830.694} C_VEL
LIN {X 0,Y 580.3,Z 260.821,A -85,B 0,C 180,E1 -1833.316,E2 -1833.316} C_VEL
LIN {X 0,Y 580.264,Z 260.833,A -85,B 0,C 180,E1 -1835.759,E2 -1835.759} C_VEL
LIN {X 0,Y 580.284,Z 260.824,A -85,B 0,C 180,E1 -1838.147,E2 -1838.147} C_VEL
LIN {X 0,Y 580.293,Z 260.821,A -85,B 0,C 180,E1 -1840.844,E2 -1840.844} C_VEL
LIN {X 0,Y 580.271,Z 260.833,A -85,B 0,C 180,E1 -1843.659,E2 -1843.659} C_VEL
LIN {X 0,Y 580.272,Z 260.823,A -85,B 0,C 180,E1 -1846.61,E2 -1846.61} C_VEL
LIN {X 0,Y 580.294,Z 260.824,A -85,B 0,C 180,E1 -1849.156,E2 -1849.156} C_VEL
LIN {X 0,Y 580.288,Z 260.825,A -85,B 0,C 180,E1 -1851.927,E2 -1851.927} C_VEL
LIN {X 0,Y 580.284,Z 260.822,A -85,B 0,C 180,E1 -1854.455,E2 -1854.455} C_VEL
LIN {X 0,Y 580.289,Z 260.824,A -85,B 0,C 180,E1 -1856.975,E2 -1856.975} C_VEL
LIN {X 0,Y 580.293,Z 260.83,A -85,B 0,C 180,E1 -1859.425,E2 -1859.425} C_VEL
LIN {X 0,Y 580.292,Z 260.824,A -85,B 0,C 180,E1 -1862.143,E2 -1862.143} C_VEL
LIN {X 0,Y 580.339,Z 260.984,A -85,B 0,C 180,E1 -1863.445,E2 -1863.445} C_VEL
LIN {X 0,Y 581.522,Z 266.955,A -85,B 0,C 180,E1 -1864.21,E2 -1864.21} C_VEL
LIN {X 0,Y 581.266,Z 291.014,A -85,B 0,C 180,E1 -1867.064,E2 -1867.064} C_VEL
LIN {X 0,Y 580.963,Z 318.021,A -85,B 0,C 180,E1 -1870.201,E2 -1870.201} C_VEL
LIN {X 0,Y 580.904,Z 321.686,A -85,B 0,C 180,E1 -1870.622,E2 -1870.622} C_VEL
LIN {X 0,Y 581.898,Z 327.364,A -85,B 0,C 180,E1 -1870.737,E2 -1870.737} C_VEL
LIN {X 0,Y 581.514,Z 488.135,A -85,B 0,C 180,E1 -1872.791,E2 -1872.791} C_VEL
LIN {X 0,Y 581.43,Z 503.717,A -85,B 0,C 180,E1 -1873.136,E2 -1873.136} C_VEL
LIN {X 0,Y 581.243,Z 519.05,A -85,B 0,C 180,E1 -1873.628,E2 -1873.628} C_VEL
LIN {X 0,Y 581.124,Z 532.775,A -85,B 0,C 180,E1 -1874.21,E2 -1874.21} C_VEL
LIN {X 0,Y 580.943,Z 546.247,A -85,B 0,C 180,E1 -1874.924,E2 -1874.924} C_VEL
LIN {X 0,Y 580.804,Z 559.484,A -85,B 0,C 180,E1 -1875.784,E2 -1875.784} C_VEL
LIN {X 0,Y 580.608,Z 571.292,A -85,B 0,C 180,E1 -1876.704,E2 -1876.704} C_VEL
LIN {X 0,Y 580.478,Z 582.752,A -85,B 0,C 180,E1 -1877.768,E2 -1877.768} C_VEL
LIN {X 0,Y 580.308,Z 593.452,A -85,B 0,C 180,E1 -1878.953,E2 -1878.953} C_VEL
LIN {X 0,Y 580.268,Z 601.859,A -85,B 0,C 180,E1 -1880.062,E2 -1880.062} C_VEL
LIN {X 0,Y 580.214,Z 609.734,A -85,B 0,C 180,E1 -1881.292,E2 -1881.292} C_VEL
LIN {X 0,Y 580.13,Z 617.09,A -85,B 0,C 180,E1 -1882.692,E2 -1882.692} C_VEL
LIN {X 0,Y 580.129,Z 622.925,A -85,B 0,C 180,E1 -1884.09,E2 -1884.09} C_VEL
LIN {X 0,Y 580.041,Z 626.386,A -85,B 0,C 180,E1 -1885.135,E2 -1885.135} C_VEL
LIN {X 0,Y 580.104,Z 629.889,A -85,B 0,C 180,E1 -1886.527,E2 -1886.527} C_VEL
LIN {X 0,Y 580.037,Z 632.193,A -85,B 0,C 180,E1 -1887.917,E2 -1887.917} C_VEL
LIN {X 0,Y 580.038,Z 633.349,A -85,B 0,C 180,E1 -1889.306,E2 -1889.306} C_VEL
LIN {X 0,Y 580.038,Z 633.349,A -85,B 0,C 180,E1 -1890.695,E2 -1890.695} C_VEL
LIN {X 0,Y 580.037,Z 632.191,A -85,B 0,C 180,E1 -1892.083,E2 -1892.083} C_VEL
LIN {X 0,Y 580.104,Z 629.886,A -85,B 0,C 180,E1 -1893.473,E2 -1893.473} C_VEL
LIN {X 0,Y 580.041,Z 626.384,A -85,B 0,C 180,E1 -1894.866,E2 -1894.866} C_VEL
LIN {X 0,Y 580.091,Z 621.607,A -85,B 0,C 180,E1 -1896.26,E2 -1896.26} C_VEL
LIN {X 0,Y 580.165,Z 615.422,A -85,B 0,C 180,E1 -1897.658,E2 -1897.658} C_VEL
LIN {X 0,Y 580.208,Z 607.647,A -85,B 0,C 180,E1 -1899.06,E2 -1899.06} C_VEL
LIN {X 0,Y 580.309,Z 599.366,A -85,B 0,C 180,E1 -1900.291,E2 -1900.291} C_VEL
LIN {X 0,Y 580.383,Z 589.391,A -85,B 0,C 180,E1 -1901.525,E2 -1901.525} C_VEL
LIN {X 0,Y 580.541,Z 579.185,A -85,B 0,C 180,E1 -1902.587,E2 -1902.587} C_VEL
LIN {X 0,Y 580.678,Z 567.014,A -85,B 0,C 180,E1 -1903.652,E2 -1903.652} C_VEL
LIN {X 0,Y 580.875,Z 553.52,A -85,B 0,C 180,E1 -1904.625,E2 -1904.625} C_VEL
LIN {X 0,Y 581.019,Z 539.861,A -85,B 0,C 180,E1 -1905.433,E2 -1905.433} C_VEL
LIN {X 0,Y 581.207,Z 525.787,A -85,B 0,C 180,E1 -1906.103,E2 -1906.103} C_VEL
LIN {X 0,Y 581.36,Z 511.291,A -85,B 0,C 180,E1 -1906.64,E2 -1906.64} C_VEL
LIN {X 0,Y 581.489,Z 496.027,A -85,B 0,C 180,E1 -1907.053,E2 -1907.053} C_VEL
LIN {X 0,Y 581.554,Z 480.487,A -85,B 0,C 180,E1 -1907.324,E2 -1907.324} C_VEL
LIN {X 0,Y 581.82,Z 326.502,A -85,B 0,C 180,E1 -1909.277,E2 -1909.277} C_VEL
LIN {X 0,Y 580.922,Z 321.536,A -85,B 0,C 180,E1 -1909.395,E2 -1909.395} C_VEL
LIN {X 0,Y 581.211,Z 295.674,A -85,B 0,C 180,E1 -1912.39,E2 -1912.39} C_VEL
LIN {X 0,Y 581.509,Z 271.737,A -85,B 0,C 180,E1 -1915.216,E2 -1915.216} C_VEL
LIN {X 0,Y 581.439,Z 265.703,A -85,B 0,C 180,E1 -1915.943,E2 -1915.943} C_VEL
LIN {X 0,Y 580.292,Z 260.831,A -85,B 0,C 180,E1 -1916.579,E2 -1916.579} C_VEL
LIN {X 0,Y 580.301,Z 260.822,A -85,B 0,C 180,E1 -1919.31,E2 -1919.31} C_VEL
LIN {X 0,Y 580.3,Z 260.825,A -85,B 0,C 180,E1 -1922.201,E2 -1922.201} C_VEL
LIN {X 0,Y 580.288,Z 260.829,A -85,B 0,C 180,E1 -1924.697,E2 -1924.697} C_VEL
LIN {X 0,Y 580.299,Z 260.82,A -85,B 0,C 180,E1 -1927.269,E2 -1927.269} C_VEL
LIN {X 0,Y 580.292,Z 260.827,A -85,B 0,C 180,E1 -1930.271,E2 -1930.271} C_VEL
LIN {X 0,Y 580.274,Z 260.828,A -85,B 0,C 180,E1 -1932.707,E2 -1932.707} C_VEL
LIN {X 0,Y 580.258,Z 260.825,A -85,B 0,C 180,E1 -1935.611,E2 -1935.611} C_VEL
LIN {X 0,Y 580.282,Z 260.83,A -85,B 0,C 180,E1 -1938.231,E2 -1938.231} C_VEL
LIN {X 0,Y 580.272,Z 260.824,A -85,B 0,C 180,E1 -1940.965,E2 -1940.965} C_VEL
LIN {X 0,Y 580.249,Z 260.827,A -85,B 0,C 180,E1 -1943.595,E2 -1943.595} C_VEL
LIN {X 0,Y 580.315,Z 260.826,A -85,B 0,C 180,E1 -1946.145,E2 -1946.145} C_VEL
LIN {X 0,Y 580.276,Z 260.826,A -85,B 0,C 180,E1 -1948.615,E2 -1948.615} C_VEL
LIN {X 0,Y 580.291,Z 260.82,A -85,B 0,C 180,E1 -1951.024,E2 -1951.024} C_VEL
LIN {X 0,Y 580.265,Z 260.833,A -85,B 0,C 180,E1 -1954.15,E2 -1954.15} C_VEL
LIN {X 0,Y 580.27,Z 260.827,A -85,B 0,C 180,E1 -1956.442,E2 -1956.442} C_VEL
LIN {X 0,Y 580.272,Z 260.824,A -85,B 0,C 180,E1 -1959.437,E2 -1959.437} C_VEL
LIN {X 0,Y 580.257,Z 260.828,A -85,B 0,C 180,E1 -1961.645,E2 -1961.645} C_VEL
LIN {X 0,Y 580.263,Z 260.831,A -85,B 0,C 180,E1 -1963.825,E2 -1963.825} C_VEL
LIN {X 0,Y 580.326,Z 260.826,A -85,B 0,C 180,E1 -1965.983,E2 -1965.983} C_VEL
LIN {X 0,Y 580.312,Z 260.817,A -85,B 0,C 180,E1 -1968.827,E2 -1968.827} C_VEL
LIN {X 0,Y 580.31,Z 260.824,A -85,B 0,C 180,E1 -1971.644,E2 -1971.644} C_VEL
LIN {X 0,Y 580.301,Z 260.822,A -85,B 0,C 180,E1 -1974.44,E2 -1974.44} C_VEL
LIN {X 0,Y 580.328,Z 260.817,A -85,B 0,C 180,E1 -1977.223,E2 -1977.223} C_VEL
LIN {X 0,Y 580.347,Z 260.821,A -85,B 0,C 180,E1 -1980,E2 -1980} C_VEL
LIN {X 0,Y 580.315,Z 260.817,A -85,B 0,C 180,E1 -1982.777,E2 -1982.777} C_VEL
LIN {X 0,Y 580.312,Z 260.825,A -85,B 0,C 180,E1 -1985.56,E2 -1985.56} C_VEL
LIN {X 0,Y 580.288,Z 260.823,A -85,B 0,C 180,E1 -1988.357,E2 -1988.357} C_VEL
LIN {X 0,Y 580.307,Z 260.82,A -85,B 0,C 180,E1 -1991.191,E2 -1991.191} C_VEL
LIN {X 0,Y 580.273,Z 260.823,A -85,B 0,C 180,E1 -1994.319,E2 -1994.319} C_VEL
LIN {X 0,Y 580.255,Z 260.826,A -85,B 0,C 180,E1 -1996.899,E2 -1996.899} C_VEL
LIN {X 0,Y 580.272,Z 260.829,A -85,B 0,C 180,E1 -1999.824,E2 -1999.824} C_VEL
LIN {X 0,Y 580.269,Z 260.829,A -85,B 0,C 180,E1 -2001.281,E2 -2001.281} C_VEL
LIN {X 0,Y 579.617,Z 260.916,A -85,B 0,C 180,E1 -2001.861,E2 -2001.861} C_VEL
LIN {X 0,Y 576.737,Z 261.275,A -85,B 0,C 180,E1 -2002.8,E2 -2002.8} C_VEL
LIN {X 0,Y 574.301,Z 261.577,A -85,B 0,C 180,E1 -2003.556,E2 -2003.556} C_VEL
LIN {X 0,Y 573.267,Z 261.698,A -85,B 0,C 180,E1 -2004.14,E2 -2004.14} C_VEL
LIN {X 0,Y 573.191,Z 261.706,A -85,B 0,C 180,E1 -2004.338,E2 -2004.338} C_VEL
LIN {X 0,Y 573.19,Z 261.707,A -85,B 0,C 180,E1 -2006.979,E2 -2006.979} C_VEL
LIN {X 0,Y 573.201,Z 261.712,A -85,B 0,C 180,E1 -2009.479,E2 -2009.479} C_VEL
LIN {X 0,Y 573.224,Z 261.701,A -85,B 0,C 180,E1 -2012.223,E2 -2012.223} C_VEL
LIN {X 0,Y 573.208,Z 261.704,A -85,B 0,C 180,E1 -2014.766,E2 -2014.766} C_VEL
LIN {X 0,Y 573.19,Z 261.708,A -85,B 0,C 180,E1 -2017.811,E2 -2017.811} C_VEL
LIN {X 0,Y 573.202,Z 261.704,A -85,B 0,C 180,E1 -2020.529,E2 -2020.529} C_VEL
LIN {X 0,Y 573.192,Z 261.714,A -85,B 0,C 180,E1 -2023.364,E2 -2023.364} C_VEL
LIN {X 0,Y 573.183,Z 261.706,A -85,B 0,C 180,E1 -2026.338,E2 -2026.338} C_VEL
LIN {X 0,Y 573.166,Z 261.709,A -85,B 0,C 180,E1 -2028.537,E2 -2028.537} C_VEL
LIN {X 0,Y 573.174,Z 261.716,A -85,B 0,C 180,E1 -2031.292,E2 -2031.292} C_VEL
LIN {X 0,Y 573.178,Z 261.707,A -85,B 0,C 180,E1 -2034.023,E2 -2034.023} C_VEL
LIN {X 0,Y 573.224,Z 261.702,A -85,B 0,C 180,E1 -2036.514,E2 -2036.514} C_VEL
LIN {X 0,Y 573.203,Z 261.714,A -85,B 0,C 180,E1 -2039.123,E2 -2039.123} C_VEL
LIN {X 0,Y 573.197,Z 261.705,A -85,B 0,C 180,E1 -2041.982,E2 -2041.982} C_VEL
LIN {X 0,Y 573.196,Z 261.709,A -85,B 0,C 180,E1 -2044.587,E2 -2044.587} C_VEL
LIN {X 0,Y 573.249,Z 261.857,A -85,B 0,C 180,E1 -2047.377,E2 -2047.377} C_VEL
LIN {X 0,Y 573.992,Z 266.456,A -85,B 0,C 180,E1 -2048.071,E2 -2048.071} C_VEL
LIN {X 0,Y 573.821,Z 283.084,A -85,B 0,C 180,E1 -2050.438,E2 -2050.438} C_VEL
LIN {X 0,Y 575.172,Z 289.915,A -85,B 0,C 180,E1 -2050.581,E2 -2050.581} C_VEL
LIN {X 0,Y 574.75,Z 448.034,A -85,B 0,C 180,E1 -2052.625,E2 -2052.625} C_VEL
LIN {X 0,Y 574.617,Z 463.731,A -85,B 0,C 180,E1 -2052.976,E2 -2052.976} C_VEL
LIN {X 0,Y 574.409,Z 479.054,A -85,B 0,C 180,E1 -2053.473,E2 -2053.473} C_VEL
LIN {X 0,Y 574.253,Z 493.716,A -85,B 0,C 180,E1 -2054.107,E2 -2054.107} C_VEL
LIN {X 0,Y 574.031,Z 507.027,A -85,B 0,C 180,E1 -2054.829,E2 -2054.829} C_VEL
LIN {X 0,Y 573.86,Z 520.549,A -85,B 0,C 180,E1 -2055.728,E2 -2055.728} C_VEL
LIN {X 0,Y 573.632,Z 532.877,A -85,B 0,C 180,E1 -2056.719,E2 -2056.719} C_VEL
LIN {X 0,Y 573.46,Z 544.075,A -85,B 0,C 180,E1 -2057.795,E2 -2057.795} C_VEL
LIN {X 0,Y 573.295,Z 553.58,A -85,B 0,C 180,E1 -2058.877,E2 -2058.877} C_VEL
LIN {X 0,Y 573.203,Z 562.774,A -85,B 0,C 180,E1 -2060.116,E2 -2060.116} C_VEL
LIN {X 0,Y 573.135,Z 570.483,A -85,B 0,C 180,E1 -2061.36,E2 -2061.36} C_VEL
LIN {X 0,Y 573.076,Z 576.881,A -85,B 0,C 180,E1 -2062.601,E2 -2062.601} C_VEL
LIN {X 0,Y 573.041,Z 582.765,A -85,B 0,C 180,E1 -2064.016,E2 -2064.016} C_VEL
LIN {X 0,Y 572.95,Z 586.249,A -85,B 0,C 180,E1 -2065.074,E2 -2065.074} C_VEL
LIN {X 0,Y 573.004,Z 589.794,A -85,B 0,C 180,E1 -2066.484,E2 -2066.484} C_VEL
LIN {X 0,Y 572.938,Z 592.139,A -85,B 0,C 180,E1 -2067.891,E2 -2067.891} C_VEL
LIN {X 0,Y 572.936,Z 593.337,A -85,B 0,C 180,E1 -2069.297,E2 -2069.297} C_VEL
LIN {X 0,Y 572.937,Z 593.359,A -85,B 0,C 180,E1 -2070.703,E2 -2070.703} C_VEL
LIN {X 0,Y 572.938,Z 592.243,A -85,B 0,C 180,E1 -2072.109,E2 -2072.109} C_VEL
LIN {X 0,Y 573.006,Z 589.982,A -85,B 0,C 180,E1 -2073.516,E2 -2073.516} C_VEL
LIN {X 0,Y 572.95,Z 586.521,A -85,B 0,C 180,E1 -2074.925,E2 -2074.925} C_VEL
LIN {X 0,Y 573.007,Z 581.789,A -85,B 0,C 180,E1 -2076.337,E2 -2076.337} C_VEL
LIN {X 0,Y 573.094,Z 575.655,A -85,B 0,C 180,E1 -2077.752,E2 -2077.752} C_VEL
LIN {X 0,Y 573.134,Z 567.935,A -85,B 0,C 180,E1 -2079.172,E2 -2079.172} C_VEL
LIN {X 0,Y 573.265,Z 559.696,A -85,B 0,C 180,E1 -2080.418,E2 -2080.418} C_VEL
LIN {X 0,Y 573.358,Z 549.787,A -85,B 0,C 180,E1 -2081.668,E2 -2081.668} C_VEL
LIN {X 0,Y 573.534,Z 539.636,A -85,B 0,C 180,E1 -2082.742,E2 -2082.742} C_VEL
LIN {X 0,Y 573.721,Z 527.558,A -85,B 0,C 180,E1 -2083.82,E2 -2083.82} C_VEL
LIN {X 0,Y 573.919,Z 514.603,A -85,B 0,C 180,E1 -2084.78,E2 -2084.78} C_VEL
LIN {X 0,Y 574.141,Z 500.721,A -85,B 0,C 180,E1 -2085.622,E2 -2085.622} C_VEL
LIN {X 0,Y 574.338,Z 485.79,A -85,B 0,C 180,E1 -2086.346,E2 -2086.346} C_VEL
LIN {X 0,Y 574.532,Z 471.278,A -85,B 0,C 180,E1 -2086.889,E2 -2086.889} C_VEL
LIN {X 0,Y 574.7,Z 455.847,A -85,B 0,C 180,E1 -2087.31,E2 -2087.31} C_VEL
LIN {X 0,Y 574.783,Z 440.788,A -85,B 0,C 180,E1 -2087.575,E2 -2087.575} C_VEL
LIN {X 0,Y 575.09,Z 289.286,A -85,B 0,C 180,E1 -2089.521,E2 -2089.521} C_VEL
LIN {X 0,Y 573.83,Z 283.086,A -85,B 0,C 180,E1 -2089.651,E2 -2089.651} C_VEL
LIN {X 0,Y 573.974,Z 265.772,A -85,B 0,C 180,E1 -2092.118,E2 -2092.118} C_VEL
LIN {X 0,Y 573.262,Z 261.705,A -85,B 0,C 180,E1 -2092.764,E2 -2092.764} C_VEL
LIN {X 0,Y 573.219,Z 261.707,A -85,B 0,C 180,E1 -2095.411,E2 -2095.411} C_VEL
LIN {X 0,Y 573.191,Z 261.71,A -85,B 0,C 180,E1 -2098.567,E2 -2098.567} C_VEL
LIN {X 0,Y 573.207,Z 261.713,A -85,B 0,C 180,E1 -2100.994,E2 -2100.994} C_VEL
LIN {X 0,Y 573.214,Z 261.705,A -85,B 0,C 180,E1 -2103.516,E2 -2103.516} C_VEL
LIN {X 0,Y 573.182,Z 261.706,A -85,B 0,C 180,E1 -2106.054,E2 -2106.054} C_VEL
LIN {X 0,Y 573.225,Z 261.709,A -85,B 0,C 180,E1 -2108.703,E2 -2108.703} C_VEL
LIN {X 0,Y 573.19,Z 261.707,A -85,B 0,C 180,E1 -2111.46,E2 -2111.46} C_VEL
LIN {X 0,Y 573.204,Z 261.706,A -85,B 0,C 180,E1 -2114.336,E2 -2114.336} C_VEL
LIN {X 0,Y 573.204,Z 261.703,A -85,B 0,C 180,E1 -2117.362,E2 -2117.362} C_VEL
LIN {X 0,Y 573.214,Z 261.71,A -85,B 0,C 180,E1 -2120.572,E2 -2120.572} C_VEL
LIN {X 0,Y 573.213,Z 261.703,A -85,B 0,C 180,E1 -2123.074,E2 -2123.074} C_VEL
LIN {X 0,Y 573.226,Z 261.7,A -85,B 0,C 180,E1 -2125.668,E2 -2125.668} C_VEL
LIN {X 0,Y 573.212,Z 261.706,A -85,B 0,C 180,E1 -2128.183,E2 -2128.183} C_VEL
LIN {X 0,Y 573.212,Z 261.712,A -85,B 0,C 180,E1 -2130.631,E2 -2130.631} C_VEL
LIN {X 0,Y 573.192,Z 261.705,A -85,B 0,C 180,E1 -2133.516,E2 -2133.516} C_VEL
LIN {X 0,Y 573.188,Z 261.709,A -85,B 0,C 180,E1 -2136.133,E2 -2136.133} C_VEL
LIN {X 0,Y 573.216,Z 261.703,A -85,B 0,C 180,E1 -2139.172,E2 -2139.172} C_VEL
LIN {X 0,Y 573.191,Z 261.704,A -85,B 0,C 180,E1 -2141.41,E2 -2141.41} C_VEL
LIN {X 0,Y 573.202,Z 261.713,A -85,B 0,C 180,E1 -2144.351,E2 -2144.351} C_VEL
LIN {X 0,Y 573.191,Z 261.713,A -85,B 0,C 180,E1 -2146.528,E2 -2146.528} C_VEL
LIN {X 0,Y 573.239,Z 261.699,A -85,B 0,C 180,E1 -2149.403,E2 -2149.403} C_VEL
LIN {X 0,Y 573.236,Z 261.708,A -85,B 0,C 180,E1 -2152.249,E2 -2152.249} C_VEL
LIN {X 0,Y 573.278,Z 261.694,A -85,B 0,C 180,E1 -2155.077,E2 -2155.077} C_VEL
LIN {X 0,Y 573.295,Z 261.696,A -85,B 0,C 180,E1 -2157.892,E2 -2157.892} C_VEL
LIN {X 0,Y 573.325,Z 261.689,A -85,B 0,C 180,E1 -2160.702,E2 -2160.702} C_VEL
LIN {X 0,Y 573.29,Z 261.694,A -85,B 0,C 180,E1 -2162.811,E2 -2162.811} C_VEL
LIN {X 0,Y 573.266,Z 261.698,A -85,B 0,C 180,E1 -2165.628,E2 -2165.628} C_VEL
LIN {X 0,Y 573.248,Z 261.702,A -85,B 0,C 180,E1 -2168.46,E2 -2168.46} C_VEL
LIN {X 0,Y 573.271,Z 261.695,A -85,B 0,C 180,E1 -2171.312,E2 -2171.312} C_VEL
LIN {X 0,Y 573.28,Z 261.697,A -85,B 0,C 180,E1 -2174.424,E2 -2174.424} C_VEL
LIN {X 0,Y 573.254,Z 261.698,A -85,B 0,C 180,E1 -2177.112,E2 -2177.112} C_VEL
LIN {X 0,Y 573.237,Z 261.708,A -85,B 0,C 180,E1 -2180.077,E2 -2180.077} C_VEL
LIN {X 0,Y 573.23,Z 261.703,A -85,B 0,C 180,E1 -2182.338,E2 -2182.338} C_VEL
LIN {X 0,Y 573.245,Z 261.698,A -85,B 0,C 180,E1 -2185.41,E2 -2185.41} C_VEL
LIN {X 0,Y 573.224,Z 261.702,A -85,B 0,C 180,E1 -2188.565,E2 -2188.565} C_VEL
LIN {X 0,Y 573.222,Z 261.7,A -85,B 0,C 180,E1 -2190.993,E2 -2190.993} C_VEL
LIN {X 0,Y 573.262,Z 261.701,A -85,B 0,C 180,E1 -2193.524,E2 -2193.524} C_VEL
LIN {X 0,Y 573.239,Z 261.703,A -85,B 0,C 180,E1 -2196.05,E2 -2196.05} C_VEL
LIN {X 0,Y 573.236,Z 261.699,A -85,B 0,C 180,E1 -2198.702,E2 -2198.702} C_VEL
LIN {X 0,Y 573.228,Z 261.71,A -85,B 0,C 180,E1 -2201.593,E2 -2201.593} C_VEL
LIN {X 0,Y 573.22,Z 261.702,A -85,B 0,C 180,E1 -2204.335,E2 -2204.335} C_VEL
LIN {X 0,Y 573.238,Z 261.705,A -85,B 0,C 180,E1 -2207.359,E2 -2207.359} C_VEL
LIN {X 0,Y 573.238,Z 261.7,A -85,B 0,C 180,E1 -2210.392,E2 -2210.392} C_VEL
LIN {X 0,Y 573.253,Z 261.701,A -85,B 0,C 180,E1 -2213.078,E2 -2213.078} C_VEL
LIN {X 0,Y 573.266,Z 261.703,A -85,B 0,C 180,E1 -2215.672,E2 -2215.672} C_VEL
LIN {X 0,Y 573.24,Z 261.701,A -85,B 0,C 180,E1 -2218.185,E2 -2218.185} C_VEL
LIN {X 0,Y 573.265,Z 261.699,A -85,B 0,C 180,E1 -2220.634,E2 -2220.634} C_VEL
LIN {X 0,Y 573.271,Z 261.825,A -85,B 0,C 180,E1 -2223.223,E2 -2223.223} C_VEL
LIN {X 0,Y 574.694,Z 268.355,A -85,B 0,C 180,E1 -2224.076,E2 -2224.076} C_VEL
LIN {X 0,Y 574.444,Z 291.444,A -85,B 0,C 180,E1 -2226.828,E2 -2226.828} C_VEL
LIN {X 0,Y 574.064,Z 318.021,A -85,B 0,C 180,E1 -2229.953,E2 -2229.953} C_VEL
LIN {X 0,Y 574.029,Z 321.72,A -85,B 0,C 180,E1 -2230.384,E2 -2230.384} C_VEL
LIN {X 0,Y 575.231,Z 328.89,A -85,B 0,C 180,E1 -2230.524,E2 -2230.524} C_VEL
LIN {X 0,Y 574.749,Z 488.296,A -85,B 0,C 180,E1 -2232.585,E2 -2232.585} C_VEL
LIN {X 0,Y 574.617,Z 503.716,A -85,B 0,C 180,E1 -2232.93,E2 -2232.93} C_VEL
LIN {X 0,Y 574.411,Z 519.047,A -85,B 0,C 180,E1 -2233.428,E2 -2233.428} C_VEL
LIN {X 0,Y 574.292,Z 532.778,A -85,B 0,C 180,E1 -2234.018,E2 -2234.018} C_VEL
LIN {X 0,Y 574.048,Z 546.25,A -85,B 0,C 180,E1 -2234.739,E2 -2234.739} C_VEL
LIN {X 0,Y 573.86,Z 559.822,A -85,B 0,C 180,E1 -2235.632,E2 -2235.632} C_VEL
LIN {X 0,Y 573.635,Z 572.353,A -85,B 0,C 180,E1 -2236.63,E2 -2236.63} C_VEL
LIN {X 0,Y 573.477,Z 582.752,A -85,B 0,C 180,E1 -2237.616,E2 -2237.616} C_VEL
LIN {X 0,Y 573.286,Z 592.771,A -85,B 0,C 180,E1 -2238.734,E2 -2238.734} C_VEL
LIN {X 0,Y 573.242,Z 601.86,A -85,B 0,C 180,E1 -2239.939,E2 -2239.939} C_VEL
LIN {X 0,Y 573.133,Z 609.735,A -85,B 0,C 180,E1 -2241.183,E2 -2241.183} C_VEL
LIN {X 0,Y 573.074,Z 617.091,A -85,B 0,C 180,E1 -2242.602,E2 -2242.602} C_VEL
LIN {X 0,Y 573.04,Z 622.924,A -85,B 0,C 180,E1 -2244.017,E2 -2244.017} C_VEL
LIN {X 0,Y 572.951,Z 626.386,A -85,B 0,C 180,E1 -2245.075,E2 -2245.075} C_VEL
LIN {X 0,Y 573.004,Z 629.89,A -85,B 0,C 180,E1 -2246.484,E2 -2246.484} C_VEL
LIN {X 0,Y 572.937,Z 632.192,A -85,B 0,C 180,E1 -2247.891,E2 -2247.891} C_VEL
LIN {X 0,Y 572.938,Z 633.349,A -85,B 0,C 180,E1 -2249.297,E2 -2249.297} C_VEL
LIN {X 0,Y 572.938,Z 633.349,A -85,B 0,C 180,E1 -2250.703,E2 -2250.703} C_VEL
LIN {X 0,Y 572.937,Z 632.19,A -85,B 0,C 180,E1 -2252.109,E2 -2252.109} C_VEL
LIN {X 0,Y 573.004,Z 629.886,A -85,B 0,C 180,E1 -2253.516,E2 -2253.516} C_VEL
LIN {X 0,Y 572.951,Z 626.384,A -85,B 0,C 180,E1 -2254.926,E2 -2254.926} C_VEL
LIN {X 0,Y 573.012,Z 621.607,A -85,B 0,C 180,E1 -2256.338,E2 -2256.338} C_VEL
LIN {X 0,Y 573.094,Z 615.421,A -85,B 0,C 180,E1 -2257.753,E2 -2257.753} C_VEL
LIN {X 0,Y 573.136,Z 607.646,A -85,B 0,C 180,E1 -2259.173,E2 -2259.173} C_VEL
LIN {X 0,Y 573.27,Z 599.366,A -85,B 0,C 180,E1 -2260.418,E2 -2260.418} C_VEL
LIN {X 0,Y 573.386,Z 589.388,A -85,B 0,C 180,E1 -2261.668,E2 -2261.668} C_VEL
LIN {X 0,Y 573.568,Z 579.185,A -85,B 0,C 180,E1 -2262.742,E2 -2262.742} C_VEL
LIN {X 0,Y 573.705,Z 567.014,A -85,B 0,C 180,E1 -2263.821,E2 -2263.821} C_VEL
LIN {X 0,Y 573.963,Z 553.897,A -85,B 0,C 180,E1 -2264.781,E2 -2264.781} C_VEL
LIN {X 0,Y 574.113,Z 541.507,A -85,B 0,C 180,E1 -2265.533,E2 -2265.533} C_VEL
LIN {X 0,Y 574.362,Z 526.822,A -85,B 0,C 180,E1 -2266.255,E2 -2266.255} C_VEL
LIN {X 0,Y 574.534,Z 512.603,A -85,B 0,C 180,E1 -2266.798,E2 -2266.798} C_VEL
LIN {X 0,Y 574.703,Z 497.567,A -85,B 0,C 180,E1 -2267.222,E2 -2267.222} C_VEL
LIN {X 0,Y 574.756,Z 482.643,A -85,B 0,C 180,E1 -2267.503,E2 -2267.503} C_VEL
LIN {X 0,Y 575.148,Z 327.633,A -85,B 0,C 180,E1 -2269.495,E2 -2269.495} C_VEL
